RoboDK station: kr30 cnc template 7 axis.rdk

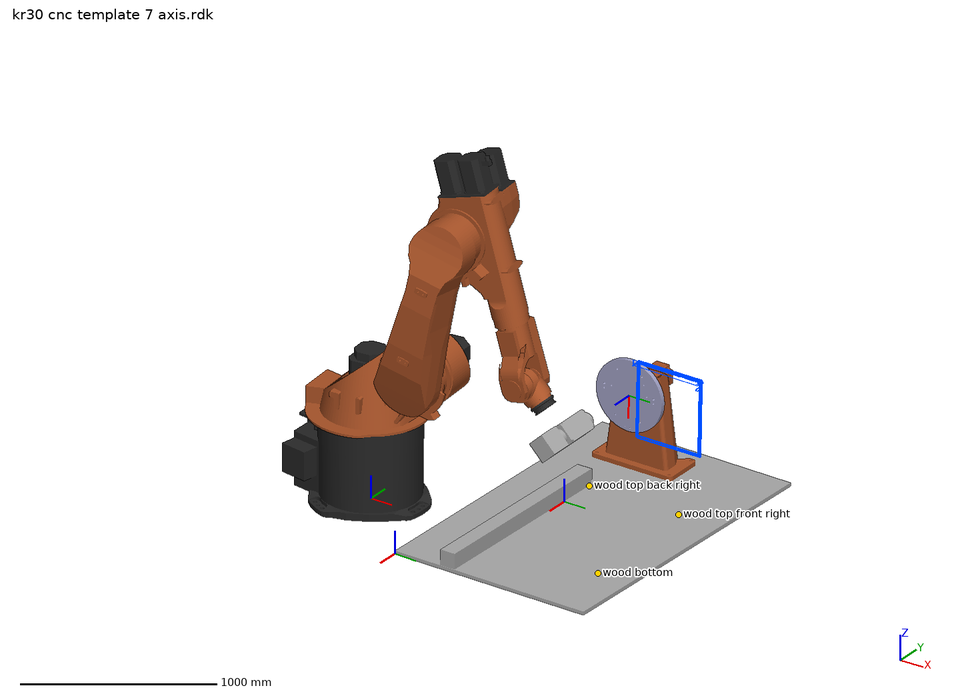
[picture v0: the station drawn from its stored meshes, robots at their saved joint values, targets as dots, program paths as lines]
Station kr30 cnc template 7 axis. Poses are relative to the parent item; angles as X-Y-Z fixed-axis rotations.
  - frame KUKA KR 30 HA Base at (0, 0, 0) mm
    - robot KUKA KR 30 HA: 6 axes, payload 30 kg, reach 2033 mm, repeatability 0.05 mm, weight 665 kg
        modified DH rows (alpha deg, a mm, theta deg, d mm): 0, 0, 0, 815; -90, 350, 0, 0; 0, 850, -90, 0; -90, 145, 0, 820; 90, 0, 0, 0; -90, 0, 180, 170
        joint limits [-185, -135, -120, -350, -119, -350] to [185, 35, 158, 350, 119, 350]; home [0, -90, 90, 0, 0, 0]; saved at [-4.811, -75.793, 150.38, -184.712, 27.792, 91.719]
      - tool rc90 spindle mm, TCP at (267.95, 0.68, 160.99) mm, rotated rx 0 ry 90 rz 0 deg, size 110 x 421.3 x 118 mm, geometry from rc90 spindle mm.stl
    - frame Tabletop at (921.82, -1104.91, 385) mm, rotated rx -0.93 ry -0.21 rz -89.9 deg
      - object tabletop CHECK HEIGHT at (-1839.9, 0, 0) mm, size 1839.9 x 1168.4 x 19 mm, geometry from kr30 tabletop mm.stl
      - object kr30 pipe jig base at (-1220, -610.6, 0) mm, size 1217.6 x 88.9 x 88.9 mm, geometry from kr30 pipe jig base.stl
      - frame Frame 3 at (-930, 400, 45) mm
      - target wood top back right (Cartesian target) at (-1141.49, 406.84, 52.26) mm, rotated rx 18.07 ry 89.88 rz 108.17 deg; joints [-2.086, -55.392, 143.759, 178.106, 87.553, -179.775] of KUKA KR 30 HA
      - target wood bottom (Cartesian target) at (-376.62, 995.52, 35.89) mm, rotated rx 18.07 ry 89.88 rz 108.17 deg; joints [24.587, -27.296, 76.752, 211.623, 53.064, -199.759] of KUKA KR 30 HA
      - target wood top front right (Cartesian target) at (-1142.68, 960.22, 52.55) mm, rotated rx 18.06 ry 89.88 rz 108.16 deg; joints [-1.42, -37.516, 98.016, 178.579, 59.693, -179.129] of KUKA KR 30 HA
  - machining project Machining Settings: C:/Users/Research Office/Desktop/paulina a5.apt | rotZ(0) | rotX(0)*rotY(0) | rotZ(0)
  - frame KUKA KP1 MD250 Base at (1360.87, 339.35, 824.43) mm, rotated rx -93.1 ry 88.62 rz 178.42 deg
    - robot KUKA KP1 MD250: 1 axes, payload 250 kg
        modified DH rows (alpha deg, a mm, theta deg, d mm): 0, 0, 0, 0
        joint limits [-180] to [180]; home [0]; saved at [179]
  - program Machining (2349 instructions, listed below)
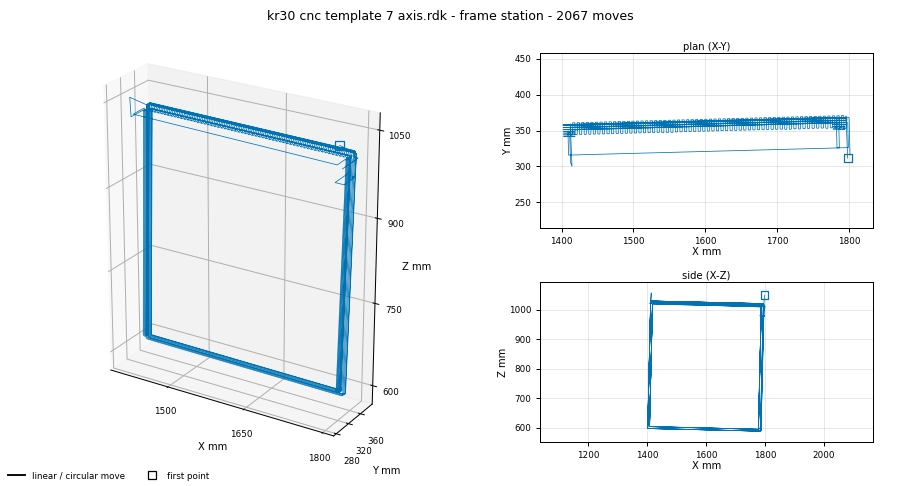
[picture p0: tool path of kr30 cnc template 7 axis.rdk in frame station, 2067 of 2067 moves have a stored position in this frame; points joined in program order, loops and branches not executed]

--- program Machining (robot KUKA KR 30 HA) ---
  Smooth(10)
  Print: /'1001'
  Print: /''
  Print: /'diagonal cut'
  Set speed (100.0 mm/s)
  Set Ref.: KUKA KP1 MD250 Base
  Set Tool: rc90 spindle mm
  Show rc90 spindle mm
  MoveJ 1 to (-235.36, 431, 39.15) mm, rotated rx 174.64 ry -29.65 rz 10.73 deg; joints [4.697, -25.984, 119.452, -143.243, 76.126, 76.923, 151.362]
  MoveL 2 to (-235.36, 431, 39.15) mm, rotated rx 174.64 ry -29.65 rz 10.73 deg; joints [4.697, -25.984, 119.452, -143.243, 76.126, 76.923, 151.362]
  MoveL 3 to (-235.36, 431, 39.15) mm, rotated rx 174.64 ry -29.65 rz 10.73 deg; joints [4.697, -25.984, 119.452, -143.243, 76.126, 76.923, 151.362]
  Set speed (100.0 mm/s)
  MoveL 4 to (-206.65, 431, -10.41) mm, rotated rx 176.37 ry -29.88 rz 7.26 deg; joints [2.395, -27.489, 120.205, -145.105, 75.237, 77.791, 154.384]
  Set speed (38.1 mm/s)
  MoveL 5 to (-201.55, 431, -19.21) mm, rotated rx 176.68 ry -29.92 rz 6.62 deg; joints [1.985, -27.751, 120.32, -145.443, 75.061, 77.953, 154.937]
  MoveL 6 to (-200.68, 431, -19.44) mm, rotated rx 176.74 ry -29.92 rz 6.52 deg; joints [1.975, -27.795, 120.334, -145.44, 75.025, 77.98, 155.032]
  Set speed (76.2 mm/s)
  MoveL 7 to (-202.44, 431, -12.48) mm, rotated rx 176.63 ry -29.91 rz 6.74 deg; joints [2.302, -27.702, 120.276, -145.137, 75.068, 77.922, 154.841]
  MoveL 8 to (-201.13, 431, -12.23) mm, rotated rx 176.71 ry -29.92 rz 6.57 deg; joints [2.315, -27.767, 120.293, -145.106, 75.011, 77.962, 154.983]
  MoveL 9 to (-196.56, 431, -16.91) mm, rotated rx 177 ry -29.95 rz 5.99 deg; joints [2.098, -27.998, 120.38, -145.259, 74.837, 78.109, 155.484]
  Set speed (38.1 mm/s)
  MoveL 10 to (-196.33, 431, -16.04) mm, rotated rx 177.01 ry -29.95 rz 5.97 deg; joints [2.14, -28.009, 120.379, -145.215, 74.823, 78.115, 155.51]
  Set speed (100.0 mm/s)
  MoveL 11 to (-203.65, 431, -3.41) mm, rotated rx 176.55 ry -29.9 rz 6.89 deg; joints [2.729, -27.635, 120.211, -144.726, 75.075, 77.876, 154.709]
  MoveL 12 to (-199.05, 427.82, -0.75) mm, rotated rx 176.75 ry -29.92 rz 6.5 deg; joints [2.857, -28.037, 120.362, -144.533, 74.826, 77.893, 155.049]
  Set speed (38.1 mm/s)
  MoveL 13 to (-197.47, 427.82, -3.47) mm, rotated rx 176.85 ry -29.93 rz 6.3 deg; joints [2.73, -28.118, 120.4, -144.638, 74.772, 77.946, 155.223]
  MoveL 14 to (-197.39, 427.82, -3.84) mm, rotated rx 176.85 ry -29.93 rz 6.29 deg; joints [2.713, -28.123, 120.403, -144.654, 74.77, 77.949, 155.232]
  Set speed (76.2 mm/s)
  MoveL 15 to (-197.71, 427.82, -8.22) mm, rotated rx 176.83 ry -29.93 rz 6.33 deg; joints [2.506, -28.11, 120.422, -144.867, 74.805, 77.944, 155.197]
  MoveL 16 to (-199.91, 427.82, -8.42) mm, rotated rx 176.69 ry -29.92 rz 6.61 deg; joints [2.494, -28, 120.393, -144.91, 74.901, 77.876, 154.954]
  MoveL 17 to (-206.05, 427.82, -11.57) mm, rotated rx 176.31 ry -29.88 rz 7.38 deg; joints [2.339, -27.694, 120.323, -145.155, 75.18, 77.69, 154.283]
  MoveL 18 to (-201.08, 427.82, -20.25) mm, rotated rx 176.62 ry -29.91 rz 6.75 deg; joints [1.934, -27.95, 120.434, -145.489, 75.005, 77.848, 154.826]
  MoveL 19 to (-201.08, 424.65, -20.25) mm, rotated rx 176.53 ry -29.9 rz 6.94 deg; joints [1.933, -28.124, 120.536, -145.493, 74.966, 77.727, 154.662]
  MoveL 20 to (-206.05, 424.65, -11.57) mm, rotated rx 176.21 ry -29.87 rz 7.57 deg; joints [2.337, -27.867, 120.426, -145.161, 75.142, 77.569, 154.116]
  MoveL 21 to (-200.05, 424.65, -8.41) mm, rotated rx 176.59 ry -29.91 rz 6.81 deg; joints [2.493, -28.167, 120.493, -144.915, 74.868, 77.75, 154.775]
  MoveL 22 to (-197.85, 424.65, -8.4) mm, rotated rx 176.73 ry -29.92 rz 6.53 deg; joints [2.496, -28.278, 120.523, -144.88, 74.772, 77.818, 155.019]
  MoveL 23 to (-197.85, 424.65, -4.14) mm, rotated rx 176.73 ry -29.92 rz 6.53 deg; joints [2.697, -28.275, 120.5, -144.678, 74.752, 77.813, 155.019]
  Set speed (38.1 mm/s)
  MoveL 24 to (-197.89, 424.65, -3.98) mm, rotated rx 176.73 ry -29.92 rz 6.54 deg; joints [2.704, -28.273, 120.498, -144.671, 74.753, 77.812, 155.014]
  MoveL 25 to (-198.05, 424.33, -3.7) mm, rotated rx 176.71 ry -29.92 rz 6.58 deg; joints [2.717, -28.282, 120.505, -144.661, 74.754, 77.794, 154.98]
  Set speed (76.2 mm/s)
  MoveL 26 to (-198.05, 421.79, -3.7) mm, rotated rx 176.63 ry -29.91 rz 6.73 deg; joints [2.716, -28.421, 120.586, -144.664, 74.722, 77.696, 154.848]
  Set speed (38.1 mm/s)
  MoveL 27 to (-197.89, 421.47, -3.98) mm, rotated rx 176.63 ry -29.91 rz 6.73 deg; joints [2.703, -28.447, 120.599, -144.674, 74.713, 77.689, 154.849]
  MoveL 28 to (-197.85, 421.47, -4.14) mm, rotated rx 176.64 ry -29.91 rz 6.72 deg; joints [2.695, -28.449, 120.601, -144.681, 74.712, 77.69, 154.854]
  Set speed (76.2 mm/s)
  MoveL 29 to (-197.85, 421.47, -8.28) mm, rotated rx 176.64 ry -29.91 rz 6.72 deg; joints [2.5, -28.452, 120.623, -144.878, 74.732, 77.696, 154.854]
  MoveL 30 to (-200, 421.47, -8.41) mm, rotated rx 176.5 ry -29.9 rz 7 deg; joints [2.492, -28.344, 120.595, -144.919, 74.826, 77.629, 154.614]
  MoveL 31 to (-206.05, 421.47, -11.57) mm, rotated rx 176.12 ry -29.85 rz 7.76 deg; joints [2.335, -28.039, 120.528, -145.168, 75.105, 77.447, 153.947]
  MoveL 32 to (-201.08, 421.47, -20.25) mm, rotated rx 176.43 ry -29.89 rz 7.13 deg; joints [1.931, -28.298, 120.638, -145.498, 74.927, 77.606, 154.495]
  MoveL 33 to (-201.08, 418.3, -20.25) mm, rotated rx 176.33 ry -29.88 rz 7.33 deg; joints [1.929, -28.471, 120.739, -145.503, 74.888, 77.483, 154.326]
  MoveL 34 to (-206.05, 418.3, -11.57) mm, rotated rx 176.02 ry -29.84 rz 7.96 deg; joints [2.333, -28.211, 120.63, -145.175, 75.068, 77.325, 153.776]
  MoveL 35 to (-199.95, 418.3, -8.41) mm, rotated rx 176.41 ry -29.89 rz 7.18 deg; joints [2.49, -28.52, 120.696, -144.922, 74.785, 77.507, 154.452]
  MoveL 36 to (-197.85, 418.3, -8.16) mm, rotated rx 176.54 ry -29.9 rz 6.91 deg; joints [2.504, -28.626, 120.723, -144.876, 74.691, 77.572, 154.687]
  MoveL 37 to (-197.85, 418.3, -4.14) mm, rotated rx 176.54 ry -29.9 rz 6.91 deg; joints [2.694, -28.623, 120.702, -144.685, 74.672, 77.567, 154.687]
  Set speed (38.1 mm/s)
  MoveL 38 to (-197.89, 418.3, -3.98) mm, rotated rx 176.54 ry -29.9 rz 6.92 deg; joints [2.701, -28.621, 120.7, -144.678, 74.673, 77.565, 154.682]
  MoveL 39 to (-198.05, 417.98, -3.7) mm, rotated rx 176.52 ry -29.9 rz 6.96 deg; joints [2.714, -28.63, 120.706, -144.668, 74.675, 77.548, 154.647]
  Set speed (76.2 mm/s)
  MoveL 40 to (-198.05, 415.44, -3.7) mm, rotated rx 176.44 ry -29.89 rz 7.11 deg; joints [2.712, -28.768, 120.787, -144.672, 74.644, 77.448, 154.512]
  Set speed (38.1 mm/s)
  MoveL 41 to (-197.89, 415.12, -3.98) mm, rotated rx 176.44 ry -29.89 rz 7.11 deg; joints [2.699, -28.794, 120.8, -144.683, 74.634, 77.441, 154.513]
  MoveL 42 to (-197.85, 415.12, -4.14) mm, rotated rx 176.44 ry -29.89 rz 7.11 deg; joints [2.692, -28.796, 120.802, -144.689, 74.633, 77.443, 154.518]
  Set speed (76.2 mm/s)
  MoveL 43 to (-197.85, 415.12, -8.4) mm, rotated rx 176.44 ry -29.89 rz 7.11 deg; joints [2.491, -28.8, 120.825, -144.892, 74.653, 77.448, 154.518]
  MoveL 44 to (-199.9, 415.12, -8.41) mm, rotated rx 176.31 ry -29.88 rz 7.37 deg; joints [2.488, -28.695, 120.798, -144.927, 74.744, 77.385, 154.288]
  MoveL 45 to (-206.05, 415.12, -11.57) mm, rotated rx 175.92 ry -29.83 rz 8.16 deg; joints [2.331, -28.382, 120.732, -145.182, 75.031, 77.201, 153.602]
  MoveL 46 to (-201.08, 415.12, -20.25) mm, rotated rx 176.24 ry -29.87 rz 7.53 deg; joints [1.927, -28.643, 120.84, -145.509, 74.849, 77.36, 154.155]
  MoveL 47 to (-201.08, 411.95, -20.25) mm, rotated rx 176.14 ry -29.86 rz 7.72 deg; joints [1.925, -28.816, 120.94, -145.515, 74.81, 77.235, 153.982]
  MoveL 48 to (-206.05, 411.95, -11.57) mm, rotated rx 175.82 ry -29.82 rz 8.36 deg; joints [2.329, -28.553, 120.833, -145.19, 74.995, 77.077, 153.427]
  MoveL 49 to (-199.84, 411.95, -8.41) mm, rotated rx 176.22 ry -29.87 rz 7.56 deg; joints [2.486, -28.87, 120.899, -144.931, 74.703, 77.262, 154.121]
  MoveL 50 to (-197.85, 411.95, -8.4) mm, rotated rx 176.35 ry -29.88 rz 7.31 deg; joints [2.489, -28.973, 120.925, -144.897, 74.614, 77.323, 154.346]
  MoveL 51 to (-197.85, 411.95, -4.14) mm, rotated rx 176.35 ry -29.88 rz 7.31 deg; joints [2.69, -28.969, 120.902, -144.694, 74.594, 77.317, 154.346]
  Set speed (38.1 mm/s)
  MoveL 52 to (-197.89, 411.95, -3.98) mm, rotated rx 176.34 ry -29.88 rz 7.31 deg; joints [2.698, -28.967, 120.9, -144.687, 74.595, 77.316, 154.342]
  MoveL 53 to (-198.05, 411.63, -3.7) mm, rotated rx 176.32 ry -29.88 rz 7.35 deg; joints [2.71, -28.976, 120.907, -144.678, 74.597, 77.298, 154.306]
  Set speed (76.2 mm/s)
  MoveL 54 to (-198.05, 409.09, -3.7) mm, rotated rx 176.24 ry -29.87 rz 7.51 deg; joints [2.709, -29.114, 120.986, -144.682, 74.566, 77.197, 154.168]
  Set speed (38.1 mm/s)
  MoveL 55 to (-197.89, 408.77, -3.98) mm, rotated rx 176.24 ry -29.87 rz 7.51 deg; joints [2.696, -29.139, 121, -144.693, 74.557, 77.19, 154.168]
  MoveL 56 to (-197.85, 408.77, -4.14) mm, rotated rx 176.25 ry -29.87 rz 7.5 deg; joints [2.688, -29.141, 121.001, -144.7, 74.555, 77.191, 154.173]
  Set speed (76.2 mm/s)
  MoveL 57 to (-197.85, 408.77, -8.4) mm, rotated rx 176.25 ry -29.87 rz 7.5 deg; joints [2.487, -29.145, 121.024, -144.903, 74.575, 77.197, 154.173]
  MoveL 58 to (-200.19, 408.77, -8.41) mm, rotated rx 176.09 ry -29.85 rz 7.81 deg; joints [2.484, -29.024, 120.994, -144.944, 74.681, 77.125, 153.907]
  MoveL 59 to (-206.05, 408.77, -11.57) mm, rotated rx 175.72 ry -29.8 rz 8.57 deg; joints [2.326, -28.724, 120.934, -145.199, 74.958, 76.952, 153.249]
  MoveL 60 to (-201.08, 408.77, -20.25) mm, rotated rx 176.04 ry -29.84 rz 7.93 deg; joints [1.923, -28.987, 121.041, -145.522, 74.772, 77.11, 153.807]
  MoveL 61 to (-201.08, 405.6, -20.25) mm, rotated rx 175.94 ry -29.83 rz 8.13 deg; joints [1.92, -29.159, 121.14, -145.53, 74.734, 76.984, 153.63]
  MoveL 62 to (-206.05, 405.6, -11.57) mm, rotated rx 175.61 ry -29.79 rz 8.77 deg; joints [2.324, -28.894, 121.035, -145.208, 74.922, 76.826, 153.069]
  MoveL 63 to (-200.12, 405.6, -8.41) mm, rotated rx 176 ry -29.84 rz 8 deg; joints [2.482, -29.199, 121.095, -144.95, 74.64, 77.001, 153.738]
  MoveL 64 to (-197.85, 405.6, -8.4) mm, rotated rx 176.15 ry -29.86 rz 7.71 deg; joints [2.485, -29.317, 121.124, -144.909, 74.536, 77.071, 153.997]
  MoveL 65 to (-197.85, 405.6, -4.14) mm, rotated rx 176.15 ry -29.86 rz 7.71 deg; joints [2.686, -29.313, 121.101, -144.706, 74.517, 77.065, 153.997]
  MoveL 66 to (-197.85, 405.47, -3.66) mm, rotated rx 176.14 ry -29.86 rz 7.71 deg; joints [2.709, -29.32, 121.102, -144.683, 74.513, 77.059, 153.99]
  MoveL 67 to (-197.85, 405.12, -3.31) mm, rotated rx 176.13 ry -29.86 rz 7.74 deg; joints [2.725, -29.338, 121.111, -144.667, 74.507, 77.044, 153.971]
  MoveL 68 to (-197.85, 404.64, -3.19) mm, rotated rx 176.12 ry -29.85 rz 7.77 deg; joints [2.731, -29.364, 121.125, -144.662, 74.501, 77.025, 153.944]
  MoveL 69 to (-197.85, 403.38, -3.19) mm, rotated rx 176.07 ry -29.85 rz 7.85 deg; joints [2.73, -29.433, 121.165, -144.665, 74.486, 76.974, 153.873]
  MoveL 70 to (-197.85, 402.9, -3.31) mm, rotated rx 176.06 ry -29.85 rz 7.88 deg; joints [2.723, -29.458, 121.18, -144.672, 74.481, 76.955, 153.846]
  MoveL 71 to (-197.85, 402.55, -3.66) mm, rotated rx 176.05 ry -29.85 rz 7.9 deg; joints [2.707, -29.477, 121.193, -144.689, 74.478, 76.941, 153.827]
  MoveL 72 to (-197.85, 402.42, -4.14) mm, rotated rx 176.04 ry -29.85 rz 7.91 deg; joints [2.684, -29.485, 121.199, -144.712, 74.479, 76.937, 153.82]
  MoveL 73 to (-197.85, 402.42, -8.4) mm, rotated rx 176.04 ry -29.85 rz 7.91 deg; joints [2.483, -29.488, 121.222, -144.915, 74.498, 76.943, 153.82]
  MoveL 74 to (-200.05, 402.42, -8.41) mm, rotated rx 175.9 ry -29.83 rz 8.2 deg; joints [2.48, -29.374, 121.195, -144.956, 74.599, 76.876, 153.567]
  MoveL 75 to (-206.05, 402.42, -11.57) mm, rotated rx 175.51 ry -29.78 rz 8.98 deg; joints [2.321, -29.063, 121.135, -145.218, 74.887, 76.699, 152.887]
  MoveL 76 to (-201.08, 402.42, -20.25) mm, rotated rx 175.83 ry -29.82 rz 8.34 deg; joints [1.918, -29.329, 121.24, -145.538, 74.697, 76.858, 153.45]
  MoveL 77 to (-201.08, 399.25, -20.25) mm, rotated rx 175.73 ry -29.81 rz 8.55 deg; joints [1.916, -29.499, 121.339, -145.547, 74.659, 76.73, 153.268]
  MoveL 78 to (-206.05, 399.25, -11.57) mm, rotated rx 175.41 ry -29.76 rz 9.2 deg; joints [2.319, -29.232, 121.235, -145.229, 74.852, 76.572, 152.702]
  MoveL 79 to (-199.98, 399.25, -8.41) mm, rotated rx 175.8 ry -29.82 rz 8.4 deg; joints [2.477, -29.548, 121.295, -144.963, 74.559, 76.75, 153.394]
  MoveL 80 to (-197.85, 399.25, -8.4) mm, rotated rx 175.94 ry -29.83 rz 8.12 deg; joints [2.481, -29.659, 121.321, -144.923, 74.46, 76.815, 153.64]
  MoveL 81 to (-197.85, 399.25, -4.14) mm, rotated rx 175.94 ry -29.83 rz 8.12 deg; joints [2.682, -29.656, 121.298, -144.72, 74.441, 76.808, 153.64]
  Set speed (38.1 mm/s)
  MoveL 82 to (-197.89, 399.25, -3.98) mm, rotated rx 175.94 ry -29.83 rz 8.12 deg; joints [2.69, -29.653, 121.297, -144.713, 74.442, 76.807, 153.635]
  MoveL 83 to (-198.05, 398.93, -3.7) mm, rotated rx 175.92 ry -29.83 rz 8.17 deg; joints [2.702, -29.662, 121.303, -144.704, 74.444, 76.789, 153.598]
  Set speed (76.2 mm/s)
  MoveL 84 to (-198.05, 396.39, -3.7) mm, rotated rx 175.83 ry -29.82 rz 8.33 deg; joints [2.7, -29.798, 121.382, -144.71, 74.415, 76.685, 153.452]
  Set speed (38.1 mm/s)
  MoveL 85 to (-197.89, 396.07, -3.98) mm, rotated rx 175.83 ry -29.82 rz 8.33 deg; joints [2.687, -29.823, 121.395, -144.721, 74.405, 76.677, 153.452]
  MoveL 86 to (-197.85, 396.07, -4.14) mm, rotated rx 175.84 ry -29.82 rz 8.33 deg; joints [2.68, -29.826, 121.396, -144.728, 74.403, 76.679, 153.457]
  Set speed (76.2 mm/s)
  MoveL 87 to (-197.85, 396.07, -8.4) mm, rotated rx 175.84 ry -29.82 rz 8.33 deg; joints [2.479, -29.829, 121.419, -144.931, 74.422, 76.686, 153.457]
  MoveL 88 to (-199.91, 396.07, -8.41) mm, rotated rx 175.7 ry -29.8 rz 8.6 deg; joints [2.475, -29.721, 121.394, -144.971, 74.518, 76.623, 153.218]
  MoveL 89 to (-206.05, 396.07, -11.57) mm, rotated rx 175.3 ry -29.75 rz 9.41 deg; joints [2.316, -29.4, 121.335, -145.241, 74.817, 76.443, 152.515]
  MoveL 90 to (-201.08, 396.07, -20.25) mm, rotated rx 175.62 ry -29.79 rz 8.76 deg; joints [1.913, -29.669, 121.438, -145.557, 74.622, 76.602, 153.084]
  MoveL 91 to (-201.08, 392.9, -20.25) mm, rotated rx 175.52 ry -29.78 rz 8.97 deg; joints [1.91, -29.838, 121.536, -145.567, 74.586, 76.473, 152.898]
  MoveL 92 to (-206.05, 392.9, -11.57) mm, rotated rx 175.19 ry -29.73 rz 9.63 deg; joints [2.313, -29.568, 121.434, -145.253, 74.782, 76.314, 152.326]
  MoveL 93 to (-199.84, 392.9, -8.41) mm, rotated rx 175.6 ry -29.79 rz 8.81 deg; joints [2.473, -29.894, 121.493, -144.979, 74.479, 76.495, 153.04]
  MoveL 94 to (-197.85, 392.9, -8.38) mm, rotated rx 175.73 ry -29.81 rz 8.54 deg; joints [2.477, -29.999, 121.517, -144.938, 74.385, 76.556, 153.272]
  MoveL 95 to (-197.85, 392.9, -4.14) mm, rotated rx 175.73 ry -29.81 rz 8.54 deg; joints [2.677, -29.996, 121.494, -144.736, 74.366, 76.549, 153.272]
  Set speed (38.1 mm/s)
  MoveL 96 to (-197.89, 392.9, -3.98) mm, rotated rx 175.73 ry -29.81 rz 8.55 deg; joints [2.685, -29.993, 121.493, -144.729, 74.368, 76.547, 153.267]
  MoveL 97 to (-198.05, 392.58, -3.7) mm, rotated rx 175.71 ry -29.8 rz 8.59 deg; joints [2.697, -30.002, 121.499, -144.72, 74.37, 76.529, 153.23]
  Set speed (76.2 mm/s)
  MoveL 98 to (-198.05, 390.04, -3.7) mm, rotated rx 175.62 ry -29.79 rz 8.76 deg; joints [2.695, -30.137, 121.577, -144.728, 74.341, 76.424, 153.08]
  Set speed (38.1 mm/s)
  MoveL 99 to (-197.89, 389.72, -3.98) mm, rotated rx 175.62 ry -29.79 rz 8.76 deg; joints [2.682, -30.162, 121.59, -144.739, 74.331, 76.416, 153.08]
  MoveL 100 to (-197.85, 389.72, -4.14) mm, rotated rx 175.62 ry -29.79 rz 8.76 deg; joints [2.675, -30.165, 121.592, -144.746, 74.329, 76.418, 153.085]
  Set speed (76.2 mm/s)
  MoveL 101 to (-197.85, 389.72, -8.26) mm, rotated rx 175.62 ry -29.79 rz 8.76 deg; joints [2.48, -30.168, 121.614, -144.942, 74.348, 76.425, 153.085]
  MoveL 102 to (-199.77, 389.72, -8.41) mm, rotated rx 175.5 ry -29.77 rz 9.01 deg; joints [2.47, -30.066, 121.592, -144.988, 74.439, 76.366, 152.86]
  MoveL 103 to (-206.05, 389.72, -11.57) mm, rotated rx 175.08 ry -29.71 rz 9.85 deg; joints [2.31, -29.736, 121.533, -145.266, 74.748, 76.184, 152.134]
  MoveL 104 to (-201.08, 389.72, -20.25) mm, rotated rx 175.41 ry -29.76 rz 9.19 deg; joints [1.908, -30.007, 121.634, -145.578, 74.549, 76.343, 152.709]
  MoveL 105 to (-201.08, 386.55, -20.25) mm, rotated rx 175.3 ry -29.75 rz 9.41 deg; joints [1.905, -30.175, 121.732, -145.59, 74.513, 76.212, 152.517]
  MoveL 106 to (-206.05, 386.55, -11.57) mm, rotated rx 174.97 ry -29.7 rz 10.07 deg; joints [2.307, -29.902, 121.632, -145.279, 74.714, 76.053, 151.94]
  MoveL 107 to (-199.7, 386.55, -8.41) mm, rotated rx 175.39 ry -29.76 rz 9.22 deg; joints [2.467, -30.238, 121.69, -144.997, 74.4, 76.237, 152.678]
  MoveL 108 to (-197.85, 386.55, -8.41) mm, rotated rx 175.52 ry -29.78 rz 8.97 deg; joints [2.471, -30.337, 121.712, -144.959, 74.312, 76.293, 152.896]
  MoveL 109 to (-197.85, 386.55, -4.14) mm, rotated rx 175.52 ry -29.78 rz 8.97 deg; joints [2.672, -30.334, 121.689, -144.756, 74.293, 76.286, 152.896]
  Set speed (38.1 mm/s)
  MoveL 110 to (-197.89, 386.55, -3.98) mm, rotated rx 175.51 ry -29.78 rz 8.98 deg; joints [2.68, -30.331, 121.688, -144.749, 74.294, 76.284, 152.89]
  MoveL 111 to (-198.05, 386.23, -3.7) mm, rotated rx 175.49 ry -29.77 rz 9.02 deg; joints [2.692, -30.339, 121.694, -144.74, 74.297, 76.266, 152.853]
  Set speed (76.2 mm/s)
  MoveL 112 to (-198.05, 383.69, -3.7) mm, rotated rx 175.4 ry -29.76 rz 9.2 deg; joints [2.69, -30.474, 121.772, -144.749, 74.268, 76.16, 152.699]
  Set speed (38.1 mm/s)
  MoveL 113 to (-197.89, 383.37, -3.98) mm, rotated rx 175.4 ry -29.76 rz 9.2 deg; joints [2.677, -30.499, 121.785, -144.76, 74.258, 76.152, 152.698]
  MoveL 114 to (-197.85, 383.37, -4.14) mm, rotated rx 175.41 ry -29.76 rz 9.19 deg; joints [2.67, -30.502, 121.786, -144.767, 74.257, 76.153, 152.703]
  Set speed (76.2 mm/s)
  MoveL 115 to (-197.85, 383.37, -8.4) mm, rotated rx 175.41 ry -29.76 rz 9.19 deg; joints [2.468, -30.505, 121.809, -144.97, 74.275, 76.161, 152.703]
  MoveL 116 to (-199.66, 383.37, -8.41) mm, rotated rx 175.28 ry -29.74 rz 9.44 deg; joints [2.465, -30.409, 121.788, -145.008, 74.362, 76.106, 152.49]
  MoveL 117 to (-206.05, 383.37, -11.57) mm, rotated rx 174.86 ry -29.68 rz 10.3 deg; joints [2.304, -30.068, 121.731, -145.294, 74.68, 75.922, 151.744]
  MoveL 118 to (-201.08, 383.37, -20.25) mm, rotated rx 175.19 ry -29.73 rz 9.63 deg; joints [1.902, -30.342, 121.83, -145.603, 74.478, 76.08, 152.323]
  MoveL 119 to (-201.08, 380.2, -20.25) mm, rotated rx 175.08 ry -29.71 rz 9.86 deg; joints [1.898, -30.509, 121.927, -145.616, 74.443, 75.947, 152.127]
  MoveL 120 to (-206.05, 380.2, -11.57) mm, rotated rx 174.75 ry -29.66 rz 10.52 deg; joints [2.3, -30.234, 121.829, -145.309, 74.647, 75.789, 151.545]
  MoveL 121 to (-200.12, 380.2, -8.41) mm, rotated rx 175.14 ry -29.72 rz 9.73 deg; joints [2.461, -30.551, 121.88, -145.03, 74.349, 75.959, 152.24]
  MoveL 122 to (-197.85, 380.2, -8.4) mm, rotated rx 175.3 ry -29.75 rz 9.42 deg; joints [2.465, -30.673, 121.906, -144.982, 74.239, 76.027, 152.509]
  MoveL 123 to (-197.85, 380.2, -4.14) mm, rotated rx 175.3 ry -29.75 rz 9.42 deg; joints [2.667, -30.669, 121.883, -144.778, 74.221, 76.02, 152.509]
  Set speed (38.1 mm/s)
  MoveL 124 to (-197.89, 380.2, -3.98) mm, rotated rx 175.29 ry -29.75 rz 9.42 deg; joints [2.674, -30.667, 121.881, -144.771, 74.223, 76.018, 152.504]
  MoveL 125 to (-198.05, 379.88, -3.7) mm, rotated rx 175.27 ry -29.74 rz 9.47 deg; joints [2.687, -30.675, 121.888, -144.763, 74.226, 75.999, 152.465]
  Set speed (76.2 mm/s)
  MoveL 126 to (-198.05, 377.34, -3.7) mm, rotated rx 175.18 ry -29.73 rz 9.65 deg; joints [2.684, -30.808, 121.965, -144.773, 74.197, 75.892, 152.307]
  Set speed (38.1 mm/s)
  MoveL 127 to (-197.89, 377.02, -3.98) mm, rotated rx 175.18 ry -29.73 rz 9.65 deg; joints [2.671, -30.834, 121.978, -144.784, 74.187, 75.884, 152.306]
  MoveL 128 to (-197.85, 377.02, -4.14) mm, rotated rx 175.18 ry -29.73 rz 9.64 deg; joints [2.664, -30.836, 121.979, -144.791, 74.186, 75.885, 152.312]
  Set speed (76.2 mm/s)
  MoveL 129 to (-197.85, 377.02, -8.4) mm, rotated rx 175.18 ry -29.73 rz 9.64 deg; joints [2.462, -30.84, 122.002, -144.994, 74.204, 75.893, 152.312]
  MoveL 130 to (-200.07, 377.02, -8.41) mm, rotated rx 175.03 ry -29.71 rz 9.95 deg; joints [2.458, -30.72, 121.978, -145.043, 74.312, 75.827, 152.048]
  MoveL 131 to (-206.05, 377.02, -11.57) mm, rotated rx 174.63 ry -29.64 rz 10.75 deg; joints [2.297, -30.399, 121.927, -145.326, 74.615, 75.656, 151.343]
  MoveL 132 to (-201.08, 377.02, -20.25) mm, rotated rx 174.96 ry -29.7 rz 10.08 deg; joints [1.895, -30.675, 122.024, -145.63, 74.408, 75.814, 151.928]
  MoveL 133 to (-201.08, 373.85, -20.25) mm, rotated rx 174.85 ry -29.68 rz 10.32 deg; joints [1.892, -30.841, 122.121, -145.646, 74.374, 75.68, 151.726]
  MoveL 134 to (-206.05, 373.85, -11.57) mm, rotated rx 174.52 ry -29.62 rz 10.99 deg; joints [2.293, -30.564, 122.025, -145.343, 74.582, 75.522, 151.138]
  MoveL 135 to (-200.58, 373.85, -8.41) mm, rotated rx 174.88 ry -29.68 rz 10.25 deg; joints [2.454, -30.858, 122.069, -145.069, 74.303, 75.677, 151.785]
  MoveL 136 to (-197.85, 373.85, -8.4) mm, rotated rx 175.07 ry -29.71 rz 9.87 deg; joints [2.459, -31.006, 122.098, -145.008, 74.169, 75.758, 152.112]
  MoveL 137 to (-197.85, 373.85, -4.14) mm, rotated rx 175.07 ry -29.71 rz 9.87 deg; joints [2.661, -31.003, 122.076, -144.804, 74.151, 75.75, 152.112]
  Set speed (38.1 mm/s)
  MoveL 138 to (-197.89, 373.85, -3.98) mm, rotated rx 175.07 ry -29.71 rz 9.88 deg; joints [2.668, -31, 122.074, -144.797, 74.153, 75.748, 152.107]
  MoveL 139 to (-198.05, 373.53, -3.7) mm, rotated rx 175.04 ry -29.71 rz 9.92 deg; joints [2.681, -31.008, 122.081, -144.789, 74.156, 75.729, 152.067]
  Set speed (76.2 mm/s)
  MoveL 140 to (-198.05, 370.99, -3.7) mm, rotated rx 174.95 ry -29.7 rz 10.11 deg; joints [2.678, -31.141, 122.157, -144.8, 74.128, 75.621, 151.905]
  Set speed (38.1 mm/s)
  MoveL 141 to (-197.89, 370.67, -3.98) mm, rotated rx 174.95 ry -29.69 rz 10.11 deg; joints [2.665, -31.166, 122.17, -144.811, 74.118, 75.612, 151.904]
  MoveL 142 to (-197.85, 370.68, -4.14) mm, rotated rx 174.95 ry -29.7 rz 10.11 deg; joints [2.658, -31.168, 122.172, -144.818, 74.117, 75.614, 151.909]
  Set speed (76.2 mm/s)
  MoveL 143 to (-197.85, 370.68, -8.4) mm, rotated rx 174.95 ry -29.7 rz 10.11 deg; joints [2.456, -31.172, 122.194, -145.022, 74.135, 75.622, 151.909]
  MoveL 144 to (-200.55, 370.67, -8.41) mm, rotated rx 174.77 ry -29.67 rz 10.48 deg; joints [2.45, -31.025, 122.166, -145.083, 74.268, 75.542, 151.585]
  MoveL 145 to (-206.05, 370.68, -11.57) mm, rotated rx 174.4 ry -29.6 rz 11.23 deg; joints [2.289, -30.727, 122.123, -145.361, 74.551, 75.387, 150.931]
  MoveL 146 to (-201.08, 370.68, -20.25) mm, rotated rx 174.73 ry -29.66 rz 10.55 deg; joints [1.888, -31.006, 122.218, -145.662, 74.34, 75.545, 151.522]
  MoveL 147 to (-201.08, 367.5, -20.25) mm, rotated rx 174.62 ry -29.64 rz 10.79 deg; joints [1.884, -31.171, 122.314, -145.679, 74.306, 75.409, 151.315]
  MoveL 148 to (-206.05, 367.5, -11.57) mm, rotated rx 174.28 ry -29.58 rz 11.47 deg; joints [2.285, -30.891, 122.22, -145.38, 74.519, 75.252, 150.722]
  MoveL 149 to (-200.51, 367.5, -8.41) mm, rotated rx 174.66 ry -29.65 rz 10.71 deg; joints [2.447, -31.192, 122.263, -145.099, 74.233, 75.407, 151.383]
  MoveL 150 to (-197.85, 367.5, -8.4) mm, rotated rx 174.84 ry -29.68 rz 10.34 deg; joints [2.453, -31.338, 122.29, -145.037, 74.1, 75.485, 151.704]
  MoveL 151 to (-197.85, 367.5, -4.14) mm, rotated rx 174.84 ry -29.68 rz 10.34 deg; joints [2.654, -31.334, 122.267, -144.833, 74.083, 75.477, 151.704]
  MoveL 152 to (-197.85, 367.37, -3.66) mm, rotated rx 174.83 ry -29.68 rz 10.35 deg; joints [2.677, -31.34, 122.269, -144.811, 74.08, 75.47, 151.696]
  MoveL 153 to (-197.85, 367.02, -3.31) mm, rotated rx 174.82 ry -29.67 rz 10.38 deg; joints [2.693, -31.358, 122.277, -144.796, 74.074, 75.455, 151.673]
  MoveL 154 to (-197.85, 366.55, -3.19) mm, rotated rx 174.8 ry -29.67 rz 10.41 deg; joints [2.698, -31.382, 122.291, -144.792, 74.069, 75.434, 151.642]
  MoveL 155 to (-197.85, 365.28, -3.19) mm, rotated rx 174.76 ry -29.66 rz 10.51 deg; joints [2.697, -31.448, 122.329, -144.799, 74.056, 75.379, 151.559]
  MoveL 156 to (-197.85, 364.8, -3.31) mm, rotated rx 174.74 ry -29.66 rz 10.54 deg; joints [2.69, -31.473, 122.344, -144.807, 74.051, 75.358, 151.527]
  MoveL 157 to (-197.85, 364.45, -3.66) mm, rotated rx 174.72 ry -29.66 rz 10.57 deg; joints [2.674, -31.491, 122.357, -144.826, 74.049, 75.344, 151.504]
  MoveL 158 to (-197.85, 364.33, -4.14) mm, rotated rx 174.72 ry -29.66 rz 10.58 deg; joints [2.651, -31.498, 122.363, -144.849, 74.05, 75.339, 151.496]
  MoveL 159 to (-197.85, 364.33, -8.4) mm, rotated rx 174.72 ry -29.66 rz 10.58 deg; joints [2.449, -31.502, 122.386, -145.053, 74.067, 75.348, 151.496]
  MoveL 160 to (-200.48, 364.33, -8.41) mm, rotated rx 174.54 ry -29.63 rz 10.94 deg; joints [2.443, -31.358, 122.359, -145.116, 74.198, 75.27, 151.177]
  MoveL 161 to (-206.05, 364.33, -11.57) mm, rotated rx 174.16 ry -29.56 rz 11.71 deg; joints [2.281, -31.053, 122.317, -145.4, 74.489, 75.115, 150.509]
  MoveL 162 to (-201.08, 364.33, -20.25) mm, rotated rx 174.5 ry -29.62 rz 11.03 deg; joints [1.881, -31.334, 122.41, -145.696, 74.274, 75.272, 151.105]
  MoveL 163 to (-201.08, 361.15, -20.25) mm, rotated rx 174.38 ry -29.6 rz 11.27 deg; joints [1.877, -31.498, 122.507, -145.715, 74.241, 75.135, 150.892]
  MoveL 164 to (-206.05, 361.15, -11.57) mm, rotated rx 174.04 ry -29.54 rz 11.96 deg; joints [2.277, -31.215, 122.415, -145.421, 74.458, 74.978, 150.294]
  MoveL 165 to (-200.44, 361.15, -8.41) mm, rotated rx 174.42 ry -29.61 rz 11.18 deg; joints [2.44, -31.523, 122.455, -145.133, 74.165, 75.133, 150.969]
  MoveL 166 to (-197.85, 361.15, -8.4) mm, rotated rx 174.6 ry -29.64 rz 10.82 deg; joints [2.445, -31.666, 122.481, -145.07, 74.034, 75.209, 151.285]
  MoveL 167 to (-197.85, 361.15, -4.14) mm, rotated rx 174.6 ry -29.64 rz 10.82 deg; joints [2.647, -31.662, 122.458, -144.866, 74.017, 75.201, 151.285]
  Set speed (38.1 mm/s)
  MoveL 168 to (-197.89, 361.15, -3.98) mm, rotated rx 174.6 ry -29.64 rz 10.83 deg; joints [2.655, -31.66, 122.457, -144.859, 74.018, 75.199, 151.28]
  MoveL 169 to (-198.05, 360.83, -3.7) mm, rotated rx 174.57 ry -29.63 rz 10.87 deg; joints [2.667, -31.667, 122.464, -144.852, 74.022, 75.18, 151.239]
  Set speed (76.2 mm/s)
  MoveL 170 to (-198.05, 358.29, -3.7) mm, rotated rx 174.48 ry -29.62 rz 11.07 deg; joints [2.664, -31.798, 122.54, -144.866, 73.996, 75.068, 151.068]
  Set speed (38.1 mm/s)
  MoveL 171 to (-197.89, 357.98, -3.98) mm, rotated rx 174.48 ry -29.62 rz 11.07 deg; joints [2.651, -31.823, 122.552, -144.877, 73.986, 75.06, 151.066]
  MoveL 172 to (-197.85, 357.98, -4.14) mm, rotated rx 174.48 ry -29.62 rz 11.07 deg; joints [2.644, -31.826, 122.554, -144.884, 73.984, 75.061, 151.072]
  Set speed (76.2 mm/s)
  MoveL 173 to (-197.85, 357.98, -8.25) mm, rotated rx 174.48 ry -29.62 rz 11.07 deg; joints [2.449, -31.829, 122.576, -145.081, 74.001, 75.07, 151.072]
  MoveL 174 to (-200.41, 357.98, -8.41) mm, rotated rx 174.3 ry -29.59 rz 11.42 deg; joints [2.436, -31.688, 122.552, -145.152, 74.131, 74.995, 150.758]
  MoveL 175 to (-206.05, 357.98, -11.57) mm, rotated rx 173.92 ry -29.52 rz 12.2 deg; joints [2.273, -31.377, 122.512, -145.443, 74.429, 74.84, 150.076]
  MoveL 176 to (-201.08, 357.98, -20.25) mm, rotated rx 174.26 ry -29.58 rz 11.52 deg; joints [1.872, -31.66, 122.602, -145.735, 74.209, 74.996, 150.677]
  MoveL 177 to (-201.08, 354.8, -20.25) mm, rotated rx 174.13 ry -29.56 rz 11.77 deg; joints [1.868, -31.822, 122.698, -145.756, 74.178, 74.857, 150.458]
  MoveL 178 to (-206.05, 354.8, -11.57) mm, rotated rx 173.79 ry -29.49 rz 12.46 deg; joints [2.268, -31.537, 122.608, -145.466, 74.399, 74.701, 149.854]
  MoveL 179 to (-200.37, 354.8, -8.41) mm, rotated rx 174.18 ry -29.57 rz 11.67 deg; joints [2.432, -31.852, 122.647, -145.171, 74.098, 74.857, 150.544]
  MoveL 180 to (-197.85, 354.8, -8.13) mm, rotated rx 174.36 ry -29.6 rz 11.31 deg; joints [2.451, -31.992, 122.67, -145.094, 73.968, 74.93, 150.855]
  MoveL 181 to (-197.85, 354.8, -4.14) mm, rotated rx 174.36 ry -29.6 rz 11.31 deg; joints [2.64, -31.988, 122.649, -144.903, 73.952, 74.921, 150.855]
  MoveL 182 to (-197.85, 354.67, -3.66) mm, rotated rx 174.35 ry -29.6 rz 11.32 deg; joints [2.662, -31.994, 122.65, -144.881, 73.949, 74.914, 150.846]
  MoveL 183 to (-197.85, 354.33, -3.31) mm, rotated rx 174.34 ry -29.59 rz 11.35 deg; joints [2.678, -32.012, 122.658, -144.866, 73.944, 74.898, 150.822]
  MoveL 184 to (-197.85, 353.85, -3.19) mm, rotated rx 174.32 ry -29.59 rz 11.39 deg; joints [2.684, -32.036, 122.672, -144.863, 73.939, 74.876, 150.789]
  MoveL 185 to (-197.85, 352.58, -3.19) mm, rotated rx 174.27 ry -29.58 rz 11.49 deg; joints [2.682, -32.101, 122.71, -144.871, 73.927, 74.82, 150.702]
  MoveL 186 to (-197.85, 352.1, -3.31) mm, rotated rx 174.25 ry -29.58 rz 11.53 deg; joints [2.675, -32.125, 122.725, -144.88, 73.922, 74.799, 150.669]
  MoveL 187 to (-197.85, 351.75, -3.66) mm, rotated rx 174.24 ry -29.58 rz 11.55 deg; joints [2.658, -32.143, 122.737, -144.899, 73.92, 74.784, 150.644]
  MoveL 188 to (-197.85, 351.63, -4.14) mm, rotated rx 174.23 ry -29.58 rz 11.56 deg; joints [2.636, -32.15, 122.744, -144.923, 73.921, 74.78, 150.635]
  MoveL 189 to (-197.85, 351.63, -8.4) mm, rotated rx 174.23 ry -29.58 rz 11.56 deg; joints [2.433, -32.154, 122.767, -145.128, 73.938, 74.789, 150.635]
  MoveL 190 to (-200.34, 351.63, -8.41) mm, rotated rx 174.06 ry -29.54 rz 11.92 deg; joints [2.427, -32.015, 122.743, -145.192, 74.066, 74.717, 150.328]
  MoveL 191 to (-206.05, 351.63, -11.57) mm, rotated rx 173.67 ry -29.47 rz 12.71 deg; joints [2.263, -31.697, 122.705, -145.491, 74.371, 74.561, 149.63]
  MoveL 192 to (-201.08, 351.63, -20.25) mm, rotated rx 174.01 ry -29.53 rz 12.02 deg; joints [1.864, -31.984, 122.794, -145.778, 74.147, 74.717, 150.237]
  MoveL 193 to (-201.08, 348.45, -20.25) mm, rotated rx 173.88 ry -29.51 rz 12.28 deg; joints [1.859, -32.144, 122.889, -145.802, 74.117, 74.576, 150.012]
  MoveL 194 to (-206.05, 348.45, -11.57) mm, rotated rx 173.54 ry -29.44 rz 12.97 deg; joints [2.258, -31.857, 122.802, -145.516, 74.342, 74.421, 149.403]
  MoveL 195 to (-199.95, 348.45, -8.41) mm, rotated rx 173.96 ry -29.53 rz 12.12 deg; joints [2.424, -32.197, 122.842, -145.204, 74.016, 74.587, 150.151]
  MoveL 196 to (-197.85, 348.45, -8.4) mm, rotated rx 174.11 ry -29.55 rz 11.82 deg; joints [2.429, -32.316, 122.861, -145.149, 73.907, 74.647, 150.413]
  MoveL 197 to (-197.85, 348.45, -4.14) mm, rotated rx 174.11 ry -29.55 rz 11.82 deg; joints [2.631, -32.312, 122.838, -144.944, 73.89, 74.638, 150.413]
  MoveL 198 to (-197.85, 348.32, -3.66) mm, rotated rx 174.1 ry -29.55 rz 11.83 deg; joints [2.654, -32.318, 122.84, -144.922, 73.887, 74.631, 150.404]
  MoveL 199 to (-197.85, 347.98, -3.31) mm, rotated rx 174.09 ry -29.55 rz 11.86 deg; joints [2.67, -32.335, 122.848, -144.908, 73.882, 74.615, 150.379]
  MoveL 200 to (-197.85, 347.5, -3.19) mm, rotated rx 174.07 ry -29.55 rz 11.9 deg; joints [2.675, -32.359, 122.862, -144.905, 73.877, 74.593, 150.345]
  MoveL 201 to (-197.85, 346.23, -3.19) mm, rotated rx 174.02 ry -29.54 rz 12 deg; joints [2.673, -32.423, 122.899, -144.914, 73.865, 74.536, 150.255]
  MoveL 202 to (-197.85, 345.75, -3.31) mm, rotated rx 174 ry -29.53 rz 12.04 deg; joints [2.667, -32.448, 122.914, -144.923, 73.861, 74.515, 150.221]
  MoveL 203 to (-197.85, 345.4, -3.66) mm, rotated rx 173.99 ry -29.53 rz 12.07 deg; joints [2.65, -32.466, 122.927, -144.943, 73.859, 74.5, 150.196]
  MoveL 204 to (-197.85, 345.28, -4.14) mm, rotated rx 173.98 ry -29.53 rz 12.08 deg; joints [2.627, -32.473, 122.933, -144.966, 73.86, 74.495, 150.187]
  MoveL 205 to (-197.85, 345.28, -8.4) mm, rotated rx 173.98 ry -29.53 rz 12.08 deg; joints [2.425, -32.477, 122.956, -145.171, 73.876, 74.505, 150.187]
  MoveL 206 to (-199.91, 345.28, -8.41) mm, rotated rx 173.84 ry -29.5 rz 12.37 deg; joints [2.419, -32.36, 122.938, -145.226, 73.984, 74.446, 149.93]
  MoveL 207 to (-206.05, 345.28, -11.57) mm, rotated rx 173.41 ry -29.42 rz 13.24 deg; joints [2.253, -32.015, 122.898, -145.543, 74.315, 74.279, 149.173]
  MoveL 208 to (-201.08, 345.28, -20.25) mm, rotated rx 173.75 ry -29.49 rz 12.54 deg; joints [1.854, -32.304, 122.984, -145.826, 74.087, 74.435, 149.785]
  MoveL 209 to (-201.08, 342.1, -20.25) mm, rotated rx 173.62 ry -29.46 rz 12.8 deg; joints [1.849, -32.464, 123.08, -145.852, 74.058, 74.292, 149.554]
  MoveL 210 to (-206.05, 342.1, -11.57) mm, rotated rx 173.28 ry -29.39 rz 13.5 deg; joints [2.248, -32.174, 122.995, -145.571, 74.288, 74.137, 148.939]
  MoveL 211 to (-199.87, 342.1, -8.41) mm, rotated rx 173.71 ry -29.48 rz 12.63 deg; joints [2.415, -32.522, 123.033, -145.25, 73.953, 74.304, 149.705]
  MoveL 212 to (-197.85, 342.1, -8.4) mm, rotated rx 173.85 ry -29.51 rz 12.34 deg; joints [2.42, -32.637, 123.051, -145.195, 73.847, 74.361, 149.958]
  MoveL 213 to (-197.85, 342.1, -4.14) mm, rotated rx 173.85 ry -29.51 rz 12.34 deg; joints [2.622, -32.633, 123.028, -144.99, 73.831, 74.351, 149.958]
  Set speed (38.1 mm/s)
  MoveL 214 to (-197.89, 342.1, -3.98) mm, rotated rx 173.85 ry -29.5 rz 12.34 deg; joints [2.63, -32.63, 123.026, -144.983, 73.832, 74.35, 149.953]
  MoveL 215 to (-198.05, 341.78, -3.7) mm, rotated rx 173.82 ry -29.5 rz 12.39 deg; joints [2.642, -32.637, 123.033, -144.977, 73.837, 74.33, 149.91]
  Set speed (76.2 mm/s)
  MoveL 216 to (-198.05, 339.25, -3.7) mm, rotated rx 173.72 ry -29.48 rz 12.61 deg; joints [2.638, -32.764, 123.109, -144.997, 73.813, 74.215, 149.724]
  Set speed (38.1 mm/s)
  MoveL 217 to (-197.89, 338.93, -3.98) mm, rotated rx 173.72 ry -29.48 rz 12.61 deg; joints [2.625, -32.789, 123.121, -145.008, 73.803, 74.205, 149.721]
  MoveL 218 to (-197.85, 338.93, -4.14) mm, rotated rx 173.72 ry -29.48 rz 12.6 deg; joints [2.618, -32.792, 123.122, -145.015, 73.802, 74.207, 149.726]
  Set speed (76.2 mm/s)
  MoveL 219 to (-197.85, 338.93, -8.4) mm, rotated rx 173.72 ry -29.48 rz 12.6 deg; joints [2.415, -32.796, 123.145, -145.22, 73.818, 74.217, 149.726]
  MoveL 220 to (-200.2, 338.93, -8.41) mm, rotated rx 173.55 ry -29.45 rz 12.94 deg; joints [2.409, -32.662, 123.125, -145.285, 73.942, 74.15, 149.43]
  MoveL 221 to (-206.05, 338.93, -11.57) mm, rotated rx 173.15 ry -29.36 rz 13.77 deg; joints [2.243, -32.331, 123.091, -145.6, 74.262, 73.994, 148.703]
  MoveL 222 to (-201.08, 338.93, -20.25) mm, rotated rx 173.49 ry -29.43 rz 13.07 deg; joints [1.844, -32.622, 123.175, -145.878, 74.03, 74.149, 149.32]
  MoveL 223 to (-201.08, 335.75, -20.25) mm, rotated rx 173.36 ry -29.41 rz 13.34 deg; joints [1.838, -32.78, 123.27, -145.906, 74.002, 74.005, 149.083]
  MoveL 224 to (-206.05, 335.75, -11.57) mm, rotated rx 173.01 ry -29.33 rz 14.04 deg; joints [2.237, -32.488, 123.187, -145.631, 74.236, 73.851, 148.463]
  MoveL 225 to (-200.15, 335.75, -8.41) mm, rotated rx 173.43 ry -29.42 rz 13.2 deg; joints [2.404, -32.823, 123.221, -145.311, 73.912, 74.007, 149.199]
  MoveL 226 to (-197.85, 335.75, -8.4) mm, rotated rx 173.59 ry -29.45 rz 12.87 deg; joints [2.41, -32.955, 123.239, -145.246, 73.789, 74.072, 149.491]
  MoveL 227 to (-197.85, 335.75, -4.14) mm, rotated rx 173.59 ry -29.45 rz 12.87 deg; joints [2.613, -32.951, 123.217, -145.041, 73.773, 74.062, 149.491]
  Set speed (38.1 mm/s)
  MoveL 228 to (-197.89, 335.75, -3.98) mm, rotated rx 173.59 ry -29.45 rz 12.88 deg; joints [2.62, -32.948, 123.215, -145.034, 73.775, 74.06, 149.485]
  MoveL 229 to (-198.05, 335.44, -3.7) mm, rotated rx 173.56 ry -29.45 rz 12.93 deg; joints [2.632, -32.955, 123.222, -145.028, 73.78, 74.04, 149.442]
  Set speed (76.2 mm/s)
  MoveL 230 to (-198.05, 332.9, -3.7) mm, rotated rx 173.45 ry -29.43 rz 13.15 deg; joints [2.628, -33.081, 123.298, -145.05, 73.758, 73.924, 149.251]
  Set speed (38.1 mm/s)
  MoveL 231 to (-197.89, 332.58, -3.98) mm, rotated rx 173.45 ry -29.43 rz 13.15 deg; joints [2.615, -33.106, 123.31, -145.061, 73.747, 73.914, 149.247]
  MoveL 232 to (-197.85, 332.58, -4.14) mm, rotated rx 173.45 ry -29.43 rz 13.14 deg; joints [2.608, -33.109, 123.311, -145.068, 73.746, 73.916, 149.252]
  Set speed (76.2 mm/s)
  MoveL 233 to (-197.85, 332.58, -8.4) mm, rotated rx 173.45 ry -29.43 rz 13.14 deg; joints [2.405, -33.113, 123.334, -145.273, 73.761, 73.926, 149.252]
  MoveL 234 to (-200.15, 332.58, -8.41) mm, rotated rx 173.29 ry -29.39 rz 13.48 deg; joints [2.398, -32.98, 123.316, -145.34, 73.885, 73.861, 148.96]
  MoveL 235 to (-206.05, 332.58, -11.57) mm, rotated rx 172.88 ry -29.3 rz 14.32 deg; joints [2.231, -32.644, 123.283, -145.662, 74.211, 73.706, 148.22]
  MoveL 236 to (-201.08, 332.58, -20.25) mm, rotated rx 173.23 ry -29.38 rz 13.61 deg; joints [1.833, -32.937, 123.365, -145.936, 73.975, 73.86, 148.843]
  MoveL 237 to (-201.08, 329.4, -20.25) mm, rotated rx 173.09 ry -29.35 rz 13.89 deg; joints [1.827, -33.094, 123.46, -145.967, 73.949, 73.714, 148.599]
  MoveL 238 to (-206.05, 329.4, -11.57) mm, rotated rx 172.74 ry -29.27 rz 14.6 deg; joints [2.225, -32.799, 123.38, -145.696, 74.186, 73.561, 147.973]
  MoveL 239 to (-200.15, 329.4, -8.41) mm, rotated rx 173.15 ry -29.36 rz 13.76 deg; joints [2.393, -33.137, 123.41, -145.37, 73.859, 73.715, 148.716]
  MoveL 240 to (-197.85, 329.4, -8.4) mm, rotated rx 173.32 ry -29.4 rz 13.42 deg; joints [2.4, -33.27, 123.428, -145.302, 73.734, 73.779, 149.01]
  MoveL 241 to (-197.85, 329.4, -4.14) mm, rotated rx 173.32 ry -29.4 rz 13.42 deg; joints [2.602, -33.266, 123.406, -145.096, 73.719, 73.769, 149.01]
  Set speed (38.1 mm/s)
  MoveL 242 to (-197.89, 329.4, -3.98) mm, rotated rx 173.32 ry -29.4 rz 13.43 deg; joints [2.61, -33.263, 123.404, -145.09, 73.72, 73.767, 149.005]
  MoveL 243 to (-198.05, 329.09, -3.7) mm, rotated rx 173.29 ry -29.39 rz 13.48 deg; joints [2.622, -33.27, 123.411, -145.084, 73.725, 73.747, 148.96]
  Set speed (76.2 mm/s)
  MoveL 244 to (-198.05, 326.55, -3.7) mm, rotated rx 173.18 ry -29.37 rz 13.7 deg; joints [2.617, -33.395, 123.487, -145.108, 73.704, 73.629, 148.764]
  Set speed (38.1 mm/s)
  MoveL 245 to (-197.89, 326.23, -3.98) mm, rotated rx 173.18 ry -29.37 rz 13.71 deg; joints [2.604, -33.42, 123.499, -145.12, 73.694, 73.619, 148.759]
  MoveL 246 to (-197.85, 326.23, -4.14) mm, rotated rx 173.18 ry -29.37 rz 13.7 deg; joints [2.597, -33.422, 123.5, -145.126, 73.692, 73.621, 148.765]
  Set speed (76.2 mm/s)
  MoveL 247 to (-197.85, 326.23, -8.4) mm, rotated rx 173.18 ry -29.37 rz 13.7 deg; joints [2.394, -33.427, 123.523, -145.332, 73.708, 73.632, 148.765]
  MoveL 248 to (-200.15, 326.23, -8.41) mm, rotated rx 173.02 ry -29.33 rz 14.04 deg; joints [2.387, -33.293, 123.505, -145.401, 73.833, 73.568, 148.469]
  MoveL 249 to (-206.05, 326.23, -11.57) mm, rotated rx 172.6 ry -29.24 rz 14.89 deg; joints [2.219, -32.953, 123.476, -145.73, 74.163, 73.415, 147.723]
  MoveL 250 to (-201.08, 326.23, -20.25) mm, rotated rx 172.95 ry -29.32 rz 14.17 deg; joints [1.821, -33.25, 123.555, -145.999, 73.923, 73.567, 148.352]
  MoveL 251 to (-201.08, 323.05, -20.25) mm, rotated rx 172.81 ry -29.29 rz 14.46 deg; joints [1.814, -33.405, 123.65, -146.033, 73.898, 73.42, 148.101]
  MoveL 252 to (-206.05, 323.05, -11.57) mm, rotated rx 172.46 ry -29.21 rz 15.17 deg; joints [2.212, -33.107, 123.572, -145.767, 74.14, 73.268, 147.47]
  MoveL 253 to (-200.15, 323.05, -8.41) mm, rotated rx 172.88 ry -29.3 rz 14.32 deg; joints [2.381, -33.448, 123.6, -145.434, 73.808, 73.42, 148.219]
  MoveL 254 to (-197.85, 323.05, -8.4) mm, rotated rx 173.04 ry -29.34 rz 13.98 deg; joints [2.388, -33.582, 123.617, -145.363, 73.682, 73.483, 148.516]
  MoveL 255 to (-197.85, 323.05, -4.14) mm, rotated rx 173.04 ry -29.34 rz 13.98 deg; joints [2.591, -33.578, 123.594, -145.158, 73.667, 73.472, 148.516]
  Set speed (38.1 mm/s)
  MoveL 256 to (-197.89, 323.05, -3.98) mm, rotated rx 173.04 ry -29.34 rz 13.99 deg; joints [2.598, -33.576, 123.593, -145.151, 73.669, 73.471, 148.51]
  MoveL 257 to (-198.05, 322.74, -3.7) mm, rotated rx 173.01 ry -29.33 rz 14.04 deg; joints [2.61, -33.582, 123.6, -145.146, 73.674, 73.451, 148.465]
  Set speed (76.2 mm/s)
  MoveL 258 to (-198.05, 320.2, -3.7) mm, rotated rx 172.9 ry -29.31 rz 14.27 deg; joints [2.606, -33.706, 123.676, -145.172, 73.654, 73.331, 148.262]
  Set speed (38.1 mm/s)
  MoveL 259 to (-197.89, 319.88, -3.98) mm, rotated rx 172.9 ry -29.31 rz 14.28 deg; joints [2.592, -33.731, 123.688, -145.184, 73.644, 73.322, 148.258]
  MoveL 260 to (-197.85, 319.88, -4.14) mm, rotated rx 172.9 ry -29.31 rz 14.27 deg; joints [2.585, -33.733, 123.689, -145.191, 73.642, 73.323, 148.263]
  Set speed (76.2 mm/s)
  MoveL 261 to (-197.85, 319.88, -8.4) mm, rotated rx 172.9 ry -29.31 rz 14.27 deg; joints [2.382, -33.738, 123.711, -145.396, 73.657, 73.334, 148.263]
  MoveL 262 to (-200.15, 319.88, -8.41) mm, rotated rx 172.74 ry -29.27 rz 14.61 deg; joints [2.375, -33.603, 123.695, -145.468, 73.784, 73.271, 147.965]
  MoveL 263 to (-206.05, 319.88, -11.57) mm, rotated rx 172.32 ry -29.17 rz 15.47 deg; joints [2.205, -33.26, 123.669, -145.804, 74.117, 73.12, 147.213]
  MoveL 264 to (-201.08, 319.88, -20.25) mm, rotated rx 172.67 ry -29.26 rz 14.75 deg; joints [1.808, -33.559, 123.745, -146.068, 73.874, 73.272, 147.846]
  MoveL 265 to (-201.08, 316.7, -20.25) mm, rotated rx 172.53 ry -29.22 rz 15.04 deg; joints [1.801, -33.713, 123.841, -146.104, 73.85, 73.122, 147.588]
  MoveL 266 to (-206.05, 316.7, -11.57) mm, rotated rx 172.17 ry -29.14 rz 15.76 deg; joints [2.198, -33.413, 123.765, -145.844, 74.096, 72.972, 146.952]
  MoveL 267 to (-200.15, 316.7, -8.41) mm, rotated rx 172.59 ry -29.24 rz 14.9 deg; joints [2.368, -33.757, 123.79, -145.504, 73.76, 73.121, 147.708]
  MoveL 268 to (-197.85, 316.7, -8.4) mm, rotated rx 172.76 ry -29.28 rz 14.56 deg; joints [2.376, -33.892, 123.806, -145.431, 73.633, 73.184, 148.007]
  MoveL 269 to (-197.85, 316.7, -4.14) mm, rotated rx 172.76 ry -29.28 rz 14.56 deg; joints [2.579, -33.888, 123.783, -145.225, 73.618, 73.173, 148.007]
  Set speed (38.1 mm/s)
  MoveL 270 to (-197.89, 316.7, -3.98) mm, rotated rx 172.76 ry -29.28 rz 14.57 deg; joints [2.586, -33.885, 123.782, -145.219, 73.62, 73.171, 148.001]
  MoveL 271 to (-198.05, 316.39, -3.7) mm, rotated rx 172.73 ry -29.27 rz 14.62 deg; joints [2.598, -33.891, 123.789, -145.214, 73.625, 73.151, 147.955]
  Set speed (76.2 mm/s)
  MoveL 272 to (-198.05, 313.85, -3.7) mm, rotated rx 172.61 ry -29.24 rz 14.86 deg; joints [2.593, -34.014, 123.865, -145.243, 73.606, 73.03, 147.747]
  Set speed (38.1 mm/s)
  MoveL 273 to (-197.89, 313.53, -3.98) mm, rotated rx 172.61 ry -29.24 rz 14.86 deg; joints [2.58, -34.039, 123.877, -145.255, 73.596, 73.02, 147.741]
  MoveL 274 to (-197.85, 313.53, -4.14) mm, rotated rx 172.62 ry -29.24 rz 14.86 deg; joints [2.572, -34.041, 123.878, -145.261, 73.594, 73.022, 147.747]
  Set speed (76.2 mm/s)
  MoveL 275 to (-197.85, 313.53, -8.4) mm, rotated rx 172.62 ry -29.24 rz 14.86 deg; joints [2.369, -34.045, 123.9, -145.467, 73.609, 73.033, 147.747]
  MoveL 276 to (-200.15, 313.53, -8.41) mm, rotated rx 172.45 ry -29.21 rz 15.2 deg; joints [2.361, -33.91, 123.885, -145.541, 73.738, 72.971, 147.446]
  MoveL 277 to (-206.05, 313.53, -11.57) mm, rotated rx 172.03 ry -29.1 rz 16.06 deg; joints [2.191, -33.564, 123.862, -145.885, 74.075, 72.823, 146.687]
  MoveL 278 to (-201.08, 313.53, -20.25) mm, rotated rx 172.38 ry -29.19 rz 15.34 deg; joints [1.794, -33.866, 123.936, -146.143, 73.827, 72.973, 147.327]
  MoveL 279 to (-201.08, 310.35, -20.25) mm, rotated rx 172.24 ry -29.15 rz 15.64 deg; joints [1.787, -34.018, 124.031, -146.183, 73.805, 72.822, 147.061]
  MoveL 280 to (-206.05, 310.35, -11.57) mm, rotated rx 171.88 ry -29.07 rz 16.36 deg; joints [2.183, -33.715, 123.958, -145.927, 74.055, 72.673, 146.419]
  MoveL 281 to (-200.15, 310.35, -8.41) mm, rotated rx 172.3 ry -29.17 rz 15.5 deg; joints [2.355, -34.062, 123.981, -145.58, 73.716, 72.82, 147.181]
  MoveL 282 to (-197.85, 310.35, -8.4) mm, rotated rx 172.47 ry -29.21 rz 15.16 deg; joints [2.363, -34.198, 123.995, -145.505, 73.586, 72.882, 147.483]
  MoveL 283 to (-197.85, 310.35, -4.14) mm, rotated rx 172.47 ry -29.21 rz 15.16 deg; joints [2.566, -34.194, 123.972, -145.299, 73.572, 72.87, 147.483]
  Set speed (38.1 mm/s)
  MoveL 284 to (-197.89, 310.35, -3.98) mm, rotated rx 172.47 ry -29.21 rz 15.16 deg; joints [2.573, -34.191, 123.971, -145.292, 73.574, 72.869, 147.478]
  MoveL 285 to (-198.05, 310.04, -3.7) mm, rotated rx 172.44 ry -29.2 rz 15.22 deg; joints [2.585, -34.197, 123.978, -145.288, 73.579, 72.848, 147.43]
  Set speed (76.2 mm/s)
  MoveL 286 to (-198.05, 307.5, -3.7) mm, rotated rx 172.32 ry -29.17 rz 15.46 deg; joints [2.579, -34.318, 124.054, -145.319, 73.562, 72.726, 147.216]
  Set speed (38.1 mm/s)
  MoveL 287 to (-197.89, 307.18, -3.98) mm, rotated rx 172.32 ry -29.17 rz 15.47 deg; joints [2.566, -34.343, 124.066, -145.331, 73.552, 72.716, 147.21]
  MoveL 288 to (-197.85, 307.18, -4.14) mm, rotated rx 172.32 ry -29.17 rz 15.46 deg; joints [2.559, -34.346, 124.067, -145.338, 73.55, 72.718, 147.216]
  Set speed (76.2 mm/s)
  MoveL 289 to (-197.85, 307.18, -8.4) mm, rotated rx 172.32 ry -29.17 rz 15.46 deg; joints [2.356, -34.35, 124.09, -145.544, 73.564, 72.729, 147.216]
  MoveL 290 to (-200.15, 307.18, -8.41) mm, rotated rx 172.15 ry -29.13 rz 15.81 deg; joints [2.347, -34.213, 124.076, -145.621, 73.695, 72.668, 146.912]
  MoveL 291 to (-206.05, 307.18, -11.57) mm, rotated rx 171.73 ry -29.03 rz 16.67 deg; joints [2.175, -33.865, 124.055, -145.972, 74.036, 72.522, 146.147]
  MoveL 292 to (-201.08, 307.18, -20.25) mm, rotated rx 172.09 ry -29.12 rz 15.94 deg; joints [1.779, -34.169, 124.127, -146.224, 73.784, 72.671, 146.792]
  MoveL 293 to (-201.08, 304.01, -20.25) mm, rotated rx 171.94 ry -29.08 rz 16.25 deg; joints [1.771, -34.319, 124.222, -146.268, 73.764, 72.518, 146.518]
  MoveL 294 to (-206.05, 304.01, -11.57) mm, rotated rx 171.58 ry -28.99 rz 16.98 deg; joints [2.167, -34.014, 124.152, -146.018, 74.017, 72.371, 145.871]
  MoveL 295 to (-200.15, 304.01, -8.41) mm, rotated rx 172 ry -29.1 rz 16.12 deg; joints [2.34, -34.364, 124.172, -145.664, 73.674, 72.515, 146.64]
  MoveL 296 to (-197.85, 304.01, -8.4) mm, rotated rx 172.17 ry -29.14 rz 15.77 deg; joints [2.348, -34.502, 124.185, -145.585, 73.543, 72.576, 146.944]
  MoveL 297 to (-197.85, 304.01, -4.14) mm, rotated rx 172.17 ry -29.14 rz 15.77 deg; joints [2.551, -34.497, 124.162, -145.379, 73.529, 72.564, 146.944]
  Set speed (38.1 mm/s)
  MoveL 298 to (-197.89, 304.01, -3.98) mm, rotated rx 172.17 ry -29.14 rz 15.78 deg; joints [2.559, -34.494, 124.161, -145.373, 73.531, 72.563, 146.938]
  MoveL 299 to (-198.05, 303.69, -3.7) mm, rotated rx 172.14 ry -29.13 rz 15.83 deg; joints [2.571, -34.5, 124.168, -145.369, 73.537, 72.542, 146.89]
  Set speed (76.2 mm/s)
  MoveL 300 to (-198.05, 301.15, -3.7) mm, rotated rx 172.02 ry -29.1 rz 16.08 deg; joints [2.565, -34.62, 124.244, -145.403, 73.521, 72.419, 146.669]
  Set speed (38.1 mm/s)
  MoveL 301 to (-197.89, 300.83, -3.98) mm, rotated rx 172.02 ry -29.1 rz 16.09 deg; joints [2.551, -34.645, 124.256, -145.415, 73.511, 72.409, 146.663]
  MoveL 302 to (-197.85, 300.83, -4.14) mm, rotated rx 172.02 ry -29.1 rz 16.08 deg; joints [2.544, -34.648, 124.257, -145.422, 73.509, 72.41, 146.669]
  Set speed (76.2 mm/s)
  MoveL 303 to (-197.85, 300.83, -8.4) mm, rotated rx 172.02 ry -29.1 rz 16.08 deg; joints [2.341, -34.652, 124.28, -145.628, 73.523, 72.422, 146.669]
  MoveL 304 to (-200.15, 300.83, -8.41) mm, rotated rx 171.85 ry -29.06 rz 16.43 deg; joints [2.332, -34.514, 124.267, -145.708, 73.655, 72.361, 146.363]
  MoveL 305 to (-206.05, 300.83, -11.57) mm, rotated rx 171.43 ry -28.95 rz 17.3 deg; joints [2.159, -34.163, 124.249, -146.066, 74, 72.219, 145.591]
  MoveL 306 to (-201.08, 300.83, -20.25) mm, rotated rx 171.78 ry -29.04 rz 16.57 deg; joints [1.763, -34.469, 124.318, -146.313, 73.744, 72.365, 146.241]
  MoveL 307 to (-201.08, 297.66, -20.25) mm, rotated rx 171.63 ry -29 rz 16.89 deg; joints [1.755, -34.618, 124.414, -146.36, 73.725, 72.212, 145.96]
  MoveL 308 to (-206.05, 297.66, -11.57) mm, rotated rx 171.27 ry -28.9 rz 17.62 deg; joints [2.15, -34.31, 124.347, -146.116, 73.983, 72.066, 145.308]
  MoveL 309 to (-200.15, 297.66, -8.41) mm, rotated rx 171.7 ry -29.02 rz 16.75 deg; joints [2.324, -34.663, 124.363, -145.754, 73.636, 72.207, 146.082]
  MoveL 310 to (-197.85, 297.66, -8.4) mm, rotated rx 171.86 ry -29.06 rz 16.4 deg; joints [2.333, -34.802, 124.375, -145.673, 73.504, 72.267, 146.389]
  MoveL 311 to (-197.85, 297.66, -4.14) mm, rotated rx 171.86 ry -29.06 rz 16.4 deg; joints [2.536, -34.797, 124.353, -145.466, 73.49, 72.255, 146.389]
  Set speed (38.1 mm/s)
  MoveL 312 to (-197.89, 297.66, -3.98) mm, rotated rx 171.86 ry -29.06 rz 16.41 deg; joints [2.544, -34.794, 124.352, -145.46, 73.492, 72.254, 146.383]
  MoveL 313 to (-198.05, 297.34, -3.7) mm, rotated rx 171.83 ry -29.05 rz 16.46 deg; joints [2.555, -34.8, 124.359, -145.457, 73.498, 72.233, 146.334]
  Set speed (76.2 mm/s)
  MoveL 314 to (-198.05, 294.8, -3.7) mm, rotated rx 171.71 ry -29.02 rz 16.72 deg; joints [2.549, -34.919, 124.435, -145.494, 73.483, 72.109, 146.107]
  Set speed (38.1 mm/s)
  MoveL 315 to (-197.89, 294.48, -3.98) mm, rotated rx 171.71 ry -29.02 rz 16.73 deg; joints [2.536, -34.943, 124.447, -145.507, 73.473, 72.098, 146.099]
  MoveL 316 to (-197.85, 294.48, -4.14) mm, rotated rx 171.71 ry -29.02 rz 16.72 deg; joints [2.528, -34.946, 124.448, -145.513, 73.471, 72.099, 146.105]
  Set speed (76.2 mm/s)
  MoveL 317 to (-197.85, 294.48, -8.4) mm, rotated rx 171.71 ry -29.02 rz 16.72 deg; joints [2.325, -34.95, 124.47, -145.72, 73.485, 72.111, 146.105]
  MoveL 318 to (-200.15, 294.48, -8.41) mm, rotated rx 171.54 ry -28.98 rz 17.07 deg; joints [2.315, -34.811, 124.459, -145.802, 73.618, 72.052, 145.797]
  MoveL 319 to (-206.05, 294.48, -11.57) mm, rotated rx 171.11 ry -28.86 rz 17.95 deg; joints [2.141, -34.457, 124.444, -146.168, 73.967, 71.912, 145.019]
  MoveL 320 to (-201.08, 294.48, -20.25) mm, rotated rx 171.47 ry -28.96 rz 17.21 deg; joints [1.746, -34.766, 124.51, -146.409, 73.707, 72.057, 145.674]
  MoveL 321 to (-201.08, 291.31, -20.25) mm, rotated rx 171.31 ry -28.91 rz 17.54 deg; joints [1.737, -34.913, 124.607, -146.46, 73.69, 71.902, 145.384]
  MoveL 322 to (-206.05, 291.31, -11.57) mm, rotated rx 170.96 ry -28.81 rz 18.28 deg; joints [2.132, -34.603, 124.542, -146.221, 73.952, 71.758, 144.727]
  MoveL 323 to (-200.15, 291.31, -8.41) mm, rotated rx 171.38 ry -28.93 rz 17.4 deg; joints [2.307, -34.958, 124.556, -145.852, 73.602, 71.896, 145.508]
  MoveL 324 to (-197.85, 291.31, -8.4) mm, rotated rx 171.55 ry -28.98 rz 17.05 deg; joints [2.316, -35.098, 124.566, -145.768, 73.468, 71.955, 145.817]
  MoveL 325 to (-197.85, 291.31, -4.14) mm, rotated rx 171.55 ry -28.98 rz 17.05 deg; joints [2.52, -35.094, 124.544, -145.561, 73.454, 71.943, 145.817]
  Set speed (38.1 mm/s)
  MoveL 326 to (-197.89, 291.31, -3.98) mm, rotated rx 171.55 ry -28.98 rz 17.05 deg; joints [2.527, -35.091, 124.543, -145.555, 73.456, 71.941, 145.811]
  MoveL 327 to (-198.05, 290.99, -3.7) mm, rotated rx 171.52 ry -28.97 rz 17.11 deg; joints [2.539, -35.096, 124.55, -145.553, 73.462, 71.921, 145.761]
  Set speed (76.2 mm/s)
  MoveL 328 to (-198.05, 288.45, -3.7) mm, rotated rx 171.39 ry -28.94 rz 17.37 deg; joints [2.532, -35.214, 124.627, -145.593, 73.449, 71.795, 145.527]
  Set speed (38.1 mm/s)
  MoveL 329 to (-197.89, 288.13, -3.98) mm, rotated rx 171.39 ry -28.93 rz 17.38 deg; joints [2.518, -35.238, 124.639, -145.606, 73.439, 71.784, 145.519]
  MoveL 330 to (-197.85, 288.13, -4.14) mm, rotated rx 171.39 ry -28.94 rz 17.38 deg; joints [2.511, -35.241, 124.64, -145.612, 73.437, 71.786, 145.525]
  Set speed (76.2 mm/s)
  MoveL 331 to (-197.85, 288.13, -8.4) mm, rotated rx 171.39 ry -28.94 rz 17.38 deg; joints [2.307, -35.246, 124.662, -145.819, 73.451, 71.798, 145.525]
  MoveL 332 to (-200.15, 288.13, -8.41) mm, rotated rx 171.22 ry -28.89 rz 17.73 deg; joints [2.298, -35.105, 124.652, -145.905, 73.586, 71.74, 145.214]
  MoveL 333 to (-206.05, 288.13, -11.57) mm, rotated rx 170.8 ry -28.77 rz 18.61 deg; joints [2.122, -34.748, 124.64, -146.277, 73.938, 71.602, 144.431]
  MoveL 334 to (-201.08, 288.13, -20.25) mm, rotated rx 171.15 ry -28.87 rz 17.87 deg; joints [1.728, -35.06, 124.704, -146.513, 73.674, 71.746, 145.09]
  MoveL 335 to (-201.08, 284.96, -20.25) mm, rotated rx 170.99 ry -28.82 rz 18.2 deg; joints [1.718, -35.205, 124.801, -146.568, 73.659, 71.589, 144.792]
  MoveL 336 to (-206.05, 284.96, -11.57) mm, rotated rx 170.63 ry -28.72 rz 18.95 deg; joints [2.112, -34.893, 124.739, -146.335, 73.925, 71.447, 144.13]
  MoveL 337 to (-200.15, 284.96, -8.41) mm, rotated rx 171.06 ry -28.84 rz 18.06 deg; joints [2.288, -35.251, 124.749, -145.959, 73.571, 71.582, 144.916]
  MoveL 338 to (-197.85, 284.96, -8.4) mm, rotated rx 171.23 ry -28.89 rz 17.71 deg; joints [2.298, -35.392, 124.759, -145.872, 73.435, 71.64, 145.228]
  MoveL 339 to (-197.85, 284.96, -4.14) mm, rotated rx 171.23 ry -28.89 rz 17.71 deg; joints [2.502, -35.387, 124.736, -145.664, 73.422, 71.628, 145.228]
  Set speed (38.1 mm/s)
  MoveL 340 to (-197.89, 284.96, -3.98) mm, rotated rx 171.23 ry -28.89 rz 17.72 deg; joints [2.509, -35.385, 124.735, -145.658, 73.424, 71.626, 145.222]
  MoveL 341 to (-198.05, 284.64, -3.7) mm, rotated rx 171.2 ry -28.88 rz 17.78 deg; joints [2.521, -35.389, 124.743, -145.656, 73.431, 71.605, 145.17]
  Set speed (76.2 mm/s)
  MoveL 342 to (-198.05, 282.1, -3.7) mm, rotated rx 171.07 ry -28.84 rz 18.05 deg; joints [2.513, -35.506, 124.82, -145.7, 73.419, 71.479, 144.929]
  Set speed (38.1 mm/s)
  MoveL 343 to (-197.89, 281.78, -3.98) mm, rotated rx 171.06 ry -28.84 rz 18.06 deg; joints [2.5, -35.53, 124.832, -145.713, 73.409, 71.467, 144.921]
  MoveL 344 to (-197.85, 281.78, -4.14) mm, rotated rx 171.06 ry -28.84 rz 18.05 deg; joints [2.493, -35.533, 124.833, -145.719, 73.407, 71.469, 144.926]
  Set speed (76.2 mm/s)
  MoveL 345 to (-197.85, 281.78, -8.4) mm, rotated rx 171.06 ry -28.84 rz 18.05 deg; joints [2.289, -35.537, 124.855, -145.927, 73.42, 71.481, 144.926]
  MoveL 346 to (-200.15, 281.78, -8.41) mm, rotated rx 170.89 ry -28.79 rz 18.4 deg; joints [2.279, -35.396, 124.846, -146.015, 73.557, 71.424, 144.613]
  MoveL 347 to (-206.05, 281.78, -11.57) mm, rotated rx 170.47 ry -28.67 rz 19.29 deg; joints [2.101, -35.036, 124.838, -146.396, 73.912, 71.29, 143.824]
  MoveL 348 to (-201.08, 281.78, -20.25) mm, rotated rx 170.83 ry -28.78 rz 18.55 deg; joints [1.708, -35.35, 124.898, -146.626, 73.645, 71.431, 144.489]
  MoveL 349 to (-201.08, 278.61, -20.25) mm, rotated rx 170.66 ry -28.73 rz 18.89 deg; joints [1.698, -35.494, 124.996, -146.686, 73.632, 71.273, 144.181]
  MoveL 350 to (-206.05, 278.61, -11.57) mm, rotated rx 170.3 ry -28.62 rz 19.64 deg; joints [2.091, -35.179, 124.937, -146.458, 73.901, 71.133, 143.515]
  MoveL 351 to (-200.15, 278.61, -8.41) mm, rotated rx 170.73 ry -28.75 rz 18.75 deg; joints [2.269, -35.54, 124.944, -146.074, 73.543, 71.265, 144.306]
  MoveL 352 to (-197.85, 278.61, -8.4) mm, rotated rx 170.9 ry -28.8 rz 18.4 deg; joints [2.279, -35.682, 124.952, -145.984, 73.406, 71.322, 144.621]
  MoveL 353 to (-197.85, 278.61, -4.14) mm, rotated rx 170.9 ry -28.8 rz 18.4 deg; joints [2.483, -35.677, 124.93, -145.776, 73.393, 71.309, 144.621]
  Set speed (38.1 mm/s)
  MoveL 354 to (-197.89, 278.61, -3.98) mm, rotated rx 170.89 ry -28.8 rz 18.4 deg; joints [2.49, -35.675, 124.929, -145.77, 73.395, 71.308, 144.615]
  MoveL 355 to (-198.05, 278.29, -3.7) mm, rotated rx 170.87 ry -28.79 rz 18.46 deg; joints [2.502, -35.679, 124.937, -145.769, 73.402, 71.287, 144.562]
  Set speed (76.2 mm/s)
  MoveL 356 to (-198.05, 275.75, -3.7) mm, rotated rx 170.73 ry -28.75 rz 18.74 deg; joints [2.494, -35.794, 125.015, -145.816, 73.392, 71.159, 144.314]
  Set speed (38.1 mm/s)
  MoveL 357 to (-197.89, 275.43, -3.98) mm, rotated rx 170.73 ry -28.75 rz 18.75 deg; joints [2.48, -35.818, 125.026, -145.829, 73.382, 71.148, 144.304]
  MoveL 358 to (-197.85, 275.43, -4.14) mm, rotated rx 170.73 ry -28.75 rz 18.75 deg; joints [2.473, -35.821, 125.027, -145.836, 73.38, 71.149, 144.31]
  Set speed (76.2 mm/s)
  MoveL 359 to (-197.85, 275.43, -8.4) mm, rotated rx 170.73 ry -28.75 rz 18.75 deg; joints [2.269, -35.826, 125.049, -146.043, 73.393, 71.162, 144.31]
  MoveL 360 to (-200.15, 275.43, -8.41) mm, rotated rx 170.56 ry -28.7 rz 19.1 deg; joints [2.258, -35.683, 125.042, -146.135, 73.531, 71.106, 143.995]
  MoveL 361 to (-206.05, 275.43, -11.57) mm, rotated rx 170.13 ry -28.56 rz 19.99 deg; joints [2.079, -35.321, 125.036, -146.523, 73.89, 70.975, 143.2]
  MoveL 362 to (-201.08, 275.43, -20.25) mm, rotated rx 170.49 ry -28.67 rz 19.24 deg; joints [1.687, -35.637, 125.094, -146.748, 73.62, 71.114, 143.869]
  MoveL 363 to (-201.08, 272.26, -20.25) mm, rotated rx 170.32 ry -28.62 rz 19.6 deg; joints [1.675, -35.779, 125.192, -146.812, 73.609, 70.954, 143.552]
  MoveL 364 to (-206.05, 272.26, -11.57) mm, rotated rx 169.96 ry -28.51 rz 20.35 deg; joints [2.068, -35.462, 125.136, -146.591, 73.881, 70.816, 142.881]
  MoveL 365 to (-200.15, 272.26, -8.41) mm, rotated rx 170.39 ry -28.64 rz 19.46 deg; joints [2.247, -35.825, 125.14, -146.198, 73.52, 70.946, 143.678]
  MoveL 366 to (-197.85, 272.26, -8.4) mm, rotated rx 170.56 ry -28.7 rz 19.1 deg; joints [2.258, -35.968, 125.147, -146.105, 73.382, 71.001, 143.995]
  MoveL 367 to (-197.85, 272.26, -4.14) mm, rotated rx 170.56 ry -28.7 rz 19.1 deg; joints [2.462, -35.964, 125.125, -145.897, 73.369, 70.988, 143.995]
  Set speed (38.1 mm/s)
  MoveL 368 to (-197.89, 272.26, -3.98) mm, rotated rx 170.56 ry -28.69 rz 19.11 deg; joints [2.47, -35.961, 125.124, -145.891, 73.371, 70.987, 143.989]
  MoveL 369 to (-198.05, 271.94, -3.7) mm, rotated rx 170.53 ry -28.69 rz 19.17 deg; joints [2.481, -35.965, 125.132, -145.891, 73.378, 70.966, 143.935]
  Set speed (76.2 mm/s)
  MoveL 370 to (-198.05, 269.4, -3.7) mm, rotated rx 170.39 ry -28.64 rz 19.46 deg; joints [2.473, -36.079, 125.211, -145.942, 73.37, 70.837, 143.679]
  Set speed (38.1 mm/s)
  MoveL 371 to (-197.89, 269.08, -3.98) mm, rotated rx 170.38 ry -28.64 rz 19.47 deg; joints [2.459, -36.103, 125.223, -145.955, 73.36, 70.825, 143.669]
  MoveL 372 to (-197.85, 269.08, -4.14) mm, rotated rx 170.39 ry -28.64 rz 19.46 deg; joints [2.452, -36.106, 125.224, -145.961, 73.358, 70.827, 143.675]
  Set speed (76.2 mm/s)
  MoveL 373 to (-197.85, 269.08, -8.4) mm, rotated rx 170.39 ry -28.64 rz 19.46 deg; joints [2.247, -36.11, 125.245, -146.169, 73.371, 70.839, 143.675]
  MoveL 374 to (-200.15, 269.08, -8.41) mm, rotated rx 170.22 ry -28.59 rz 19.82 deg; joints [2.236, -35.967, 125.239, -146.264, 73.51, 70.785, 143.357]
  MoveL 375 to (-206.05, 269.08, -11.57) mm, rotated rx 169.79 ry -28.45 rz 20.71 deg; joints [2.056, -35.602, 125.237, -146.661, 73.873, 70.657, 142.557]
  MoveL 376 to (-201.08, 269.08, -20.25) mm, rotated rx 170.15 ry -28.57 rz 19.96 deg; joints [1.664, -35.92, 125.291, -146.879, 73.598, 70.794, 143.23]
  MoveL 377 to (-201.08, 265.91, -20.25) mm, rotated rx 169.97 ry -28.51 rz 20.33 deg; joints [1.652, -36.06, 125.391, -146.948, 73.589, 70.632, 142.904]
  MoveL 378 to (-206.05, 265.91, -11.57) mm, rotated rx 169.61 ry -28.39 rz 21.08 deg; joints [2.043, -35.741, 125.338, -146.733, 73.865, 70.497, 142.228]
  MoveL 379 to (-200.15, 265.91, -8.41) mm, rotated rx 170.04 ry -28.53 rz 20.18 deg; joints [2.225, -36.107, 125.339, -146.333, 73.501, 70.623, 143.031]
  MoveL 380 to (-197.85, 265.91, -8.4) mm, rotated rx 170.21 ry -28.59 rz 19.83 deg; joints [2.236, -36.252, 125.344, -146.236, 73.361, 70.677, 143.349]
  MoveL 381 to (-197.85, 265.91, -4.14) mm, rotated rx 170.21 ry -28.59 rz 19.83 deg; joints [2.44, -36.247, 125.322, -146.028, 73.348, 70.664, 143.349]
  Set speed (38.1 mm/s)
  MoveL 382 to (-197.89, 265.91, -3.98) mm, rotated rx 170.21 ry -28.59 rz 19.83 deg; joints [2.448, -36.244, 125.321, -146.022, 73.35, 70.663, 143.344]
  MoveL 383 to (-198.05, 265.59, -3.7) mm, rotated rx 170.18 ry -28.58 rz 19.89 deg; joints [2.459, -36.248, 125.33, -146.022, 73.358, 70.642, 143.289]
  Set speed (76.2 mm/s)
  MoveL 384 to (-198.05, 263.05, -3.7) mm, rotated rx 170.04 ry -28.53 rz 20.19 deg; joints [2.45, -36.36, 125.409, -146.078, 73.351, 70.512, 143.024]
  Set speed (38.1 mm/s)
  MoveL 385 to (-197.89, 262.73, -3.98) mm, rotated rx 170.03 ry -28.53 rz 20.2 deg; joints [2.436, -36.384, 125.421, -146.091, 73.342, 70.5, 143.013]
  MoveL 386 to (-197.85, 262.73, -4.14) mm, rotated rx 170.03 ry -28.53 rz 20.2 deg; joints [2.429, -36.387, 125.422, -146.097, 73.34, 70.501, 143.019]
  Set speed (76.2 mm/s)
  MoveL 387 to (-197.85, 262.73, -8.4) mm, rotated rx 170.03 ry -28.53 rz 20.2 deg; joints [2.224, -36.392, 125.443, -146.305, 73.352, 70.514, 143.019]
  MoveL 388 to (-200.15, 262.73, -8.41) mm, rotated rx 169.86 ry -28.47 rz 20.55 deg; joints [2.213, -36.247, 125.439, -146.404, 73.493, 70.461, 142.7]
  MoveL 389 to (-206.05, 262.73, -11.57) mm, rotated rx 169.44 ry -28.33 rz 21.45 deg; joints [2.031, -35.879, 125.439, -146.808, 73.859, 70.337, 141.895]
  MoveL 390 to (-201.08, 262.73, -20.25) mm, rotated rx 169.8 ry -28.45 rz 20.7 deg; joints [1.639, -36.2, 125.491, -147.02, 73.581, 70.471, 142.572]
  MoveL 391 to (-201.08, 259.56, -20.25) mm, rotated rx 169.62 ry -28.39 rz 21.07 deg; joints [1.626, -36.338, 125.591, -147.095, 73.574, 70.308, 142.235]
  MoveL 392 to (-206.05, 259.56, -11.57) mm, rotated rx 169.26 ry -28.27 rz 21.83 deg; joints [2.017, -36.016, 125.541, -146.886, 73.853, 70.175, 141.556]
  MoveL 393 to (-200.15, 259.56, -8.41) mm, rotated rx 169.68 ry -28.42 rz 20.93 deg; joints [2.2, -36.386, 125.539, -146.477, 73.486, 70.298, 142.363]
  MoveL 394 to (-197.85, 259.56, -8.4) mm, rotated rx 169.86 ry -28.47 rz 20.57 deg; joints [2.212, -36.531, 125.543, -146.377, 73.344, 70.351, 142.684]
  MoveL 395 to (-197.85, 259.56, -4.14) mm, rotated rx 169.86 ry -28.47 rz 20.57 deg; joints [2.417, -36.526, 125.521, -146.169, 73.332, 70.338, 142.684]
  Set speed (38.1 mm/s)
  MoveL 396 to (-197.89, 259.56, -3.98) mm, rotated rx 169.85 ry -28.47 rz 20.58 deg; joints [2.424, -36.524, 125.521, -146.163, 73.334, 70.336, 142.678]
  MoveL 397 to (-198.05, 259.24, -3.7) mm, rotated rx 169.82 ry -28.46 rz 20.64 deg; joints [2.435, -36.527, 125.529, -146.164, 73.342, 70.315, 142.622]
  Set speed (76.2 mm/s)
  MoveL 398 to (-198.05, 256.7, -3.7) mm, rotated rx 169.68 ry -28.41 rz 20.95 deg; joints [2.425, -36.638, 125.609, -146.224, 73.337, 70.184, 142.35]
  Set speed (38.1 mm/s)
  MoveL 399 to (-197.89, 256.38, -3.98) mm, rotated rx 169.67 ry -28.41 rz 20.96 deg; joints [2.412, -36.662, 125.621, -146.238, 73.328, 70.172, 142.338]
  MoveL 400 to (-197.85, 256.38, -4.14) mm, rotated rx 169.67 ry -28.41 rz 20.95 deg; joints [2.404, -36.665, 125.622, -146.244, 73.326, 70.173, 142.344]
  Set speed (76.2 mm/s)
  MoveL 401 to (-197.85, 256.38, -8.4) mm, rotated rx 169.67 ry -28.41 rz 20.95 deg; joints [2.199, -36.669, 125.643, -146.452, 73.338, 70.186, 142.344]
  MoveL 402 to (-200.15, 256.38, -8.41) mm, rotated rx 169.5 ry -28.35 rz 21.31 deg; joints [2.187, -36.523, 125.64, -146.554, 73.48, 70.134, 142.022]
  MoveL 403 to (-206.05, 256.38, -11.57) mm, rotated rx 169.08 ry -28.2 rz 22.22 deg; joints [2.004, -36.153, 125.644, -146.966, 73.849, 70.014, 141.212]
  MoveL 404 to (-201.08, 256.38, -20.25) mm, rotated rx 169.44 ry -28.33 rz 21.46 deg; joints [1.613, -36.476, 125.692, -147.172, 73.568, 70.145, 141.894]
  MoveL 405 to (-201.08, 253.21, -20.25) mm, rotated rx 169.25 ry -28.27 rz 21.84 deg; joints [1.599, -36.613, 125.794, -147.253, 73.563, 69.981, 141.546]
  MoveL 406 to (-206.05, 253.21, -11.57) mm, rotated rx 168.89 ry -28.14 rz 22.61 deg; joints [1.989, -36.289, 125.747, -147.05, 73.846, 69.851, 140.863]
  MoveL 407 to (-200.15, 253.21, -8.41) mm, rotated rx 169.32 ry -28.29 rz 21.7 deg; joints [2.174, -36.66, 125.742, -146.633, 73.475, 69.97, 141.675]
  MoveL 408 to (-197.85, 253.21, -8.4) mm, rotated rx 169.49 ry -28.35 rz 21.34 deg; joints [2.186, -36.807, 125.744, -146.53, 73.332, 70.021, 141.998]
  MoveL 409 to (-197.85, 253.21, -4.14) mm, rotated rx 169.49 ry -28.35 rz 21.34 deg; joints [2.391, -36.802, 125.723, -146.322, 73.32, 70.008, 141.998]
  Set speed (38.1 mm/s)
  MoveL 410 to (-197.89, 253.21, -3.98) mm, rotated rx 169.49 ry -28.35 rz 21.35 deg; joints [2.399, -36.799, 125.722, -146.316, 73.322, 70.007, 141.992]
  MoveL 411 to (-198.05, 252.89, -3.7) mm, rotated rx 169.46 ry -28.34 rz 21.41 deg; joints [2.41, -36.803, 125.731, -146.317, 73.331, 69.986, 141.934]
  Set speed (76.2 mm/s)
  MoveL 412 to (-198.05, 250.35, -3.7) mm, rotated rx 169.31 ry -28.29 rz 21.72 deg; joints [2.399, -36.912, 125.812, -146.382, 73.328, 69.853, 141.653]
  Set speed (38.1 mm/s)
  MoveL 413 to (-197.89, 250.03, -3.98) mm, rotated rx 169.3 ry -28.28 rz 21.74 deg; joints [2.385, -36.936, 125.824, -146.396, 73.318, 69.841, 141.64]
  MoveL 414 to (-197.85, 250.03, -4.14) mm, rotated rx 169.3 ry -28.28 rz 21.73 deg; joints [2.378, -36.939, 125.825, -146.402, 73.316, 69.842, 141.646]
  Set speed (76.2 mm/s)
  MoveL 415 to (-197.85, 250.03, -8.4) mm, rotated rx 169.3 ry -28.28 rz 21.73 deg; joints [2.173, -36.943, 125.846, -146.611, 73.328, 69.856, 141.646]
  MoveL 416 to (-200.15, 250.03, -8.41) mm, rotated rx 169.13 ry -28.22 rz 22.09 deg; joints [2.16, -36.796, 125.844, -146.715, 73.471, 69.805, 141.323]
  MoveL 417 to (-206.05, 250.03, -11.57) mm, rotated rx 168.71 ry -28.07 rz 23 deg; joints [1.975, -36.423, 125.851, -147.136, 73.843, 69.688, 140.509]
  MoveL 418 to (-201.08, 250.03, -20.25) mm, rotated rx 169.07 ry -28.2 rz 22.24 deg; joints [1.585, -36.748, 125.896, -147.336, 73.559, 69.817, 141.194]
  MoveL 419 to (-201.08, 246.86, -20.25) mm, rotated rx 168.88 ry -28.13 rz 22.64 deg; joints [1.57, -36.883, 125.999, -147.422, 73.557, 69.652, 140.836]
  MoveL 420 to (-206.05, 246.86, -11.57) mm, rotated rx 168.52 ry -28 rz 23.4 deg; joints [1.959, -36.557, 125.955, -147.226, 73.842, 69.525, 140.149]
  MoveL 421 to (-200.15, 246.86, -8.41) mm, rotated rx 168.95 ry -28.16 rz 22.49 deg; joints [2.145, -36.931, 125.947, -146.801, 73.469, 69.64, 140.965]
  MoveL 422 to (-197.85, 246.86, -8.4) mm, rotated rx 169.12 ry -28.22 rz 22.13 deg; joints [2.159, -37.079, 125.948, -146.694, 73.325, 69.689, 141.29]
  MoveL 423 to (-197.85, 246.86, -4.14) mm, rotated rx 169.12 ry -28.22 rz 22.13 deg; joints [2.364, -37.074, 125.927, -146.486, 73.313, 69.676, 141.29]
  Set speed (38.1 mm/s)
  MoveL 424 to (-197.89, 246.86, -3.98) mm, rotated rx 169.11 ry -28.22 rz 22.14 deg; joints [2.371, -37.071, 125.926, -146.48, 73.315, 69.675, 141.284]
  MoveL 425 to (-198.05, 246.54, -3.7) mm, rotated rx 169.08 ry -28.21 rz 22.2 deg; joints [2.382, -37.075, 125.935, -146.482, 73.324, 69.654, 141.225]
  Set speed (76.2 mm/s)
  MoveL 426 to (-198.05, 244, -3.7) mm, rotated rx 168.93 ry -28.15 rz 22.52 deg; joints [2.37, -37.182, 126.017, -146.552, 73.322, 69.52, 140.935]
  Set speed (38.1 mm/s)
  MoveL 427 to (-197.89, 243.69, -3.98) mm, rotated rx 168.92 ry -28.15 rz 22.54 deg; joints [2.357, -37.206, 126.029, -146.566, 73.313, 69.508, 140.921]
  MoveL 428 to (-197.85, 243.69, -4.14) mm, rotated rx 168.93 ry -28.15 rz 22.53 deg; joints [2.349, -37.209, 126.03, -146.572, 73.311, 69.509, 140.927]
  Set speed (76.2 mm/s)
  MoveL 429 to (-197.85, 243.69, -8.4) mm, rotated rx 168.93 ry -28.15 rz 22.53 deg; joints [2.144, -37.214, 126.051, -146.781, 73.323, 69.523, 140.927]
  MoveL 430 to (-200.15, 243.69, -8.41) mm, rotated rx 168.75 ry -28.09 rz 22.9 deg; joints [2.13, -37.066, 126.05, -146.889, 73.467, 69.473, 140.602]
  MoveL 431 to (-206.05, 243.69, -11.57) mm, rotated rx 168.33 ry -27.92 rz 23.8 deg; joints [1.944, -36.69, 126.06, -147.318, 73.842, 69.361, 139.784]
  MoveL 432 to (-201.08, 243.69, -20.25) mm, rotated rx 168.69 ry -28.06 rz 23.04 deg; joints [1.554, -37.017, 126.103, -147.512, 73.555, 69.486, 140.472]
  MoveL 433 to (-201.08, 240.51, -20.25) mm, rotated rx 168.49 ry -27.99 rz 23.45 deg; joints [1.538, -37.15, 126.207, -147.604, 73.555, 69.32, 140.103]
  MoveL 434 to (-206.05, 240.51, -11.57) mm, rotated rx 168.14 ry -27.85 rz 24.21 deg; joints [1.927, -36.822, 126.166, -147.414, 73.843, 69.196, 139.413]
  MoveL 435 to (-200.15, 240.51, -8.41) mm, rotated rx 168.56 ry -28.01 rz 23.31 deg; joints [2.115, -37.199, 126.155, -146.981, 73.467, 69.307, 140.233]
  MoveL 436 to (-197.85, 240.51, -8.4) mm, rotated rx 168.73 ry -28.08 rz 22.94 deg; joints [2.129, -37.347, 126.155, -146.871, 73.322, 69.355, 140.559]
  MoveL 437 to (-197.85, 240.51, -4.14) mm, rotated rx 168.73 ry -28.08 rz 22.94 deg; joints [2.334, -37.343, 126.134, -146.662, 73.31, 69.342, 140.559]
  Set speed (38.1 mm/s)
  MoveL 438 to (-197.89, 240.51, -3.98) mm, rotated rx 168.73 ry -28.08 rz 22.95 deg; joints [2.342, -37.34, 126.133, -146.656, 73.312, 69.34, 140.553]
  MoveL 439 to (-198.05, 240.19, -3.7) mm, rotated rx 168.7 ry -28.06 rz 23.02 deg; joints [2.352, -37.343, 126.142, -146.66, 73.322, 69.319, 140.493]
  Set speed (76.2 mm/s)
  MoveL 440 to (-198.05, 237.65, -3.7) mm, rotated rx 168.54 ry -28.01 rz 23.35 deg; joints [2.34, -37.449, 126.226, -146.734, 73.322, 69.185, 140.194]
  Set speed (38.1 mm/s)
  MoveL 441 to (-197.89, 237.34, -3.98) mm, rotated rx 168.53 ry -28 rz 23.37 deg; joints [2.326, -37.473, 126.238, -146.749, 73.313, 69.172, 140.179]
  MoveL 442 to (-197.85, 237.34, -4.14) mm, rotated rx 168.54 ry -28 rz 23.36 deg; joints [2.319, -37.475, 126.238, -146.755, 73.31, 69.174, 140.185]
  Set speed (76.2 mm/s)
  MoveL 443 to (-197.85, 237.34, -8.4) mm, rotated rx 168.54 ry -28 rz 23.36 deg; joints [2.113, -37.48, 126.26, -146.964, 73.322, 69.187, 140.185]
  MoveL 444 to (-200.15, 237.34, -8.41) mm, rotated rx 168.37 ry -27.94 rz 23.72 deg; joints [2.099, -37.331, 126.26, -147.076, 73.468, 69.14, 139.858]
  MoveL 445 to (-206.05, 237.34, -11.57) mm, rotated rx 167.94 ry -27.77 rz 24.63 deg; joints [1.91, -36.953, 126.273, -147.513, 73.845, 69.031, 139.036]
  MoveL 446 to (-201.08, 237.34, -20.25) mm, rotated rx 168.3 ry -27.91 rz 23.87 deg; joints [1.522, -37.282, 126.312, -147.701, 73.555, 69.153, 139.728]
  MoveL 447 to (-201.08, 234.16, -20.25) mm, rotated rx 168.1 ry -27.83 rz 24.29 deg; joints [1.505, -37.413, 126.418, -147.8, 73.557, 68.985, 139.347]
  MoveL 448 to (-206.05, 234.16, -11.57) mm, rotated rx 167.75 ry -27.69 rz 25.05 deg; joints [1.893, -37.083, 126.38, -147.616, 73.849, 68.865, 138.654]
  MoveL 449 to (-200.15, 234.16, -8.41) mm, rotated rx 168.17 ry -27.86 rz 24.14 deg; joints [2.082, -37.462, 126.366, -147.174, 73.47, 68.972, 139.477]
  MoveL 450 to (-197.85, 234.16, -8.4) mm, rotated rx 168.34 ry -27.93 rz 23.78 deg; joints [2.097, -37.612, 126.365, -147.061, 73.323, 69.018, 139.805]
  MoveL 451 to (-197.85, 234.16, -4.14) mm, rotated rx 168.34 ry -27.93 rz 23.78 deg; joints [2.302, -37.607, 126.344, -146.852, 73.312, 69.005, 139.805]
  Set speed (38.1 mm/s)
  MoveL 452 to (-197.89, 234.16, -3.98) mm, rotated rx 168.34 ry -27.93 rz 23.79 deg; joints [2.31, -37.604, 126.343, -146.846, 73.314, 69.004, 139.799]
  MoveL 453 to (-198.05, 233.84, -3.7) mm, rotated rx 168.3 ry -27.91 rz 23.85 deg; joints [2.32, -37.607, 126.352, -146.85, 73.324, 68.983, 139.738]
  Set speed (76.2 mm/s)
  MoveL 454 to (-198.05, 231.3, -3.7) mm, rotated rx 168.14 ry -27.85 rz 24.2 deg; joints [2.307, -37.712, 126.437, -146.93, 73.326, 68.847, 139.429]
  Set speed (38.1 mm/s)
  MoveL 455 to (-197.89, 230.99, -3.98) mm, rotated rx 168.14 ry -27.85 rz 24.21 deg; joints [2.293, -37.735, 126.449, -146.946, 73.317, 68.835, 139.413]
  MoveL 456 to (-197.85, 230.99, -4.14) mm, rotated rx 168.14 ry -27.85 rz 24.21 deg; joints [2.286, -37.738, 126.45, -146.952, 73.315, 68.836, 139.419]
  Set speed (76.2 mm/s)
  MoveL 457 to (-197.85, 230.99, -8.4) mm, rotated rx 168.14 ry -27.85 rz 24.21 deg; joints [2.08, -37.743, 126.471, -147.161, 73.326, 68.849, 139.419]
  MoveL 458 to (-200.15, 230.99, -8.41) mm, rotated rx 167.97 ry -27.78 rz 24.57 deg; joints [2.065, -37.593, 126.473, -147.276, 73.473, 68.803, 139.091]
  MoveL 459 to (-206.05, 230.99, -11.57) mm, rotated rx 167.55 ry -27.61 rz 25.48 deg; joints [1.875, -37.212, 126.489, -147.722, 73.853, 68.699, 138.266]
  MoveL 460 to (-201.08, 230.99, -20.25) mm, rotated rx 167.9 ry -27.75 rz 24.72 deg; joints [1.487, -37.544, 126.525, -147.903, 73.56, 68.817, 138.96]
  MoveL 461 to (-201.08, 227.81, -20.25) mm, rotated rx 167.7 ry -27.67 rz 25.15 deg; joints [1.469, -37.673, 126.633, -148.01, 73.565, 68.649, 138.567]
  MoveL 462 to (-206.05, 227.81, -11.57) mm, rotated rx 167.35 ry -27.52 rz 25.92 deg; joints [1.856, -37.34, 126.598, -147.832, 73.859, 68.532, 137.872]
  MoveL 463 to (-200.15, 227.81, -8.41) mm, rotated rx 167.77 ry -27.7 rz 25 deg; joints [2.047, -37.722, 126.581, -147.382, 73.477, 68.635, 138.698]
  MoveL 464 to (-197.85, 227.81, -8.4) mm, rotated rx 167.94 ry -27.77 rz 24.64 deg; joints [2.062, -37.873, 126.578, -147.265, 73.33, 68.68, 139.027]
  MoveL 465 to (-197.85, 227.81, -4.14) mm, rotated rx 167.94 ry -27.77 rz 24.64 deg; joints [2.268, -37.868, 126.557, -147.056, 73.319, 68.666, 139.027]
  Set speed (38.1 mm/s)
  MoveL 466 to (-197.89, 227.81, -3.98) mm, rotated rx 167.93 ry -27.77 rz 24.65 deg; joints [2.276, -37.865, 126.557, -147.05, 73.321, 68.665, 139.021]
  MoveL 467 to (-198.05, 227.49, -3.7) mm, rotated rx 167.9 ry -27.75 rz 24.72 deg; joints [2.286, -37.867, 126.566, -147.055, 73.331, 68.644, 138.958]
  Set speed (76.2 mm/s)
  MoveL 468 to (-198.05, 224.95, -3.7) mm, rotated rx 167.74 ry -27.69 rz 25.07 deg; joints [2.272, -37.971, 126.653, -147.141, 73.335, 68.508, 138.64]
  Set speed (38.1 mm/s)
  MoveL 469 to (-197.89, 224.64, -3.98) mm, rotated rx 167.73 ry -27.68 rz 25.09 deg; joints [2.258, -37.994, 126.665, -147.157, 73.326, 68.495, 138.622]
  MoveL 470 to (-197.85, 224.64, -4.14) mm, rotated rx 167.73 ry -27.68 rz 25.08 deg; joints [2.25, -37.997, 126.666, -147.163, 73.324, 68.496, 138.629]
  Set speed (76.2 mm/s)
  MoveL 471 to (-197.85, 224.64, -8.4) mm, rotated rx 167.73 ry -27.68 rz 25.08 deg; joints [2.044, -38.001, 126.686, -147.373, 73.335, 68.509, 138.629]
  MoveL 472 to (-200.15, 224.64, -8.41) mm, rotated rx 167.56 ry -27.61 rz 25.45 deg; joints [2.029, -37.851, 126.689, -147.491, 73.483, 68.465, 138.299]
  MoveL 473 to (-206.05, 224.64, -11.57) mm, rotated rx 167.14 ry -27.43 rz 26.36 deg; joints [1.836, -37.468, 126.708, -147.945, 73.866, 68.365, 137.471]
  MoveL 474 to (-201.08, 224.64, -20.25) mm, rotated rx 167.5 ry -27.58 rz 25.59 deg; joints [1.449, -37.801, 126.742, -148.12, 73.57, 68.48, 138.168]
  MoveL 475 to (-201.08, 221.46, -20.25) mm, rotated rx 167.29 ry -27.5 rz 26.04 deg; joints [1.43, -37.928, 126.851, -148.234, 73.577, 68.31, 137.762]
  MoveL 476 to (-206.05, 221.46, -11.57) mm, rotated rx 166.94 ry -27.34 rz 26.8 deg; joints [1.816, -37.594, 126.82, -148.062, 73.874, 68.198, 137.065]
  MoveL 477 to (-200.15, 221.46, -8.41) mm, rotated rx 167.36 ry -27.53 rz 25.89 deg; joints [2.01, -37.978, 126.799, -147.604, 73.49, 68.296, 137.893]
  MoveL 478 to (-197.85, 221.46, -8.4) mm, rotated rx 167.53 ry -27.6 rz 25.53 deg; joints [2.025, -38.129, 126.795, -147.484, 73.341, 68.339, 138.224]
  MoveL 479 to (-197.85, 221.46, -4.14) mm, rotated rx 167.53 ry -27.6 rz 25.53 deg; joints [2.232, -38.125, 126.775, -147.274, 73.33, 68.325, 138.224]
  Set speed (38.1 mm/s)
  MoveL 480 to (-197.89, 221.46, -3.98) mm, rotated rx 167.52 ry -27.6 rz 25.53 deg; joints [2.239, -38.122, 126.774, -147.269, 73.333, 68.324, 138.218]
  MoveL 481 to (-198.05, 221.14, -3.7) mm, rotated rx 167.49 ry -27.58 rz 25.6 deg; joints [2.249, -38.124, 126.784, -147.275, 73.343, 68.303, 138.154]
  Set speed (76.2 mm/s)
  MoveL 482 to (-198.05, 218.6, -3.7) mm, rotated rx 167.32 ry -27.51 rz 25.97 deg; joints [2.234, -38.226, 126.872, -147.367, 73.349, 68.166, 137.825]
  Set speed (38.1 mm/s)
  MoveL 483 to (-197.89, 218.29, -3.98) mm, rotated rx 167.31 ry -27.51 rz 25.99 deg; joints [2.22, -38.249, 126.884, -147.384, 73.34, 68.153, 137.806]
  MoveL 484 to (-197.85, 218.29, -4.14) mm, rotated rx 167.32 ry -27.51 rz 25.98 deg; joints [2.212, -38.252, 126.885, -147.389, 73.338, 68.154, 137.812]
  Set speed (76.2 mm/s)
  MoveL 485 to (-197.85, 218.29, -8.4) mm, rotated rx 167.32 ry -27.51 rz 25.98 deg; joints [2.006, -38.256, 126.906, -147.6, 73.349, 68.168, 137.812]
  MoveL 486 to (-200.15, 218.29, -8.41) mm, rotated rx 167.15 ry -27.43 rz 26.34 deg; joints [1.99, -38.105, 126.91, -147.721, 73.498, 68.125, 137.482]
  MoveL 487 to (-206.05, 218.29, -11.57) mm, rotated rx 166.73 ry -27.25 rz 27.25 deg; joints [1.795, -37.719, 126.932, -148.184, 73.883, 68.03, 136.652]
  MoveL 488 to (-201.08, 218.29, -20.25) mm, rotated rx 167.08 ry -27.4 rz 26.49 deg; joints [1.409, -38.055, 126.962, -148.352, 73.585, 68.14, 137.35]
  MoveL 489 to (-201.08, 215.11, -20.25) mm, rotated rx 166.87 ry -27.31 rz 26.95 deg; joints [1.388, -38.18, 127.074, -148.474, 73.594, 67.97, 136.931]
  MoveL 490 to (-206.05, 215.11, -11.57) mm, rotated rx 166.52 ry -27.15 rz 27.71 deg; joints [1.774, -37.844, 127.045, -148.309, 73.893, 67.862, 136.233]
  MoveL 491 to (-200.15, 215.11, -8.41) mm, rotated rx 166.94 ry -27.34 rz 26.8 deg; joints [1.969, -38.23, 127.022, -147.842, 73.507, 67.955, 137.063]
  MoveL 492 to (-197.85, 215.11, -8.4) mm, rotated rx 167.1 ry -27.41 rz 26.44 deg; joints [1.986, -38.383, 127.017, -147.719, 73.358, 67.996, 137.394]
  MoveL 493 to (-197.85, 215.11, -4.14) mm, rotated rx 167.1 ry -27.41 rz 26.44 deg; joints [2.192, -38.378, 126.996, -147.509, 73.347, 67.983, 137.394]
  Set speed (38.1 mm/s)
  MoveL 494 to (-197.89, 215.11, -3.98) mm, rotated rx 167.1 ry -27.41 rz 26.45 deg; joints [2.2, -38.375, 126.996, -147.503, 73.349, 67.982, 137.388]
  MoveL 495 to (-198.05, 214.79, -3.7) mm, rotated rx 167.07 ry -27.4 rz 26.52 deg; joints [2.21, -38.377, 127.006, -147.51, 73.36, 67.961, 137.323]
  Set speed (76.2 mm/s)
  MoveL 496 to (-198.05, 212.26, -3.7) mm, rotated rx 166.9 ry -27.32 rz 26.89 deg; joints [2.193, -38.477, 127.096, -147.609, 73.368, 67.823, 136.983]
  Set speed (38.1 mm/s)
  MoveL 497 to (-197.89, 211.94, -3.98) mm, rotated rx 166.89 ry -27.32 rz 26.91 deg; joints [2.179, -38.5, 127.108, -147.627, 73.359, 67.81, 136.963]
  MoveL 498 to (-197.85, 211.94, -4.14) mm, rotated rx 166.89 ry -27.32 rz 26.91 deg; joints [2.171, -38.503, 127.109, -147.632, 73.357, 67.811, 136.97]
  Set speed (76.2 mm/s)
  MoveL 499 to (-197.85, 211.94, -8.4) mm, rotated rx 166.89 ry -27.32 rz 26.91 deg; joints [1.965, -38.508, 127.129, -147.843, 73.368, 67.824, 136.97]
  MoveL 500 to (-200.15, 211.94, -8.41) mm, rotated rx 166.72 ry -27.24 rz 27.27 deg; joints [1.948, -38.355, 127.135, -147.967, 73.517, 67.784, 136.638]
  MoveL 501 to (-206.05, 211.94, -11.57) mm, rotated rx 166.31 ry -27.05 rz 28.18 deg; joints [1.751, -37.967, 127.159, -148.438, 73.904, 67.693, 135.807]
  MoveL 502 to (-201.08, 211.94, -20.25) mm, rotated rx 166.66 ry -27.21 rz 27.41 deg; joints [1.366, -38.304, 127.186, -148.601, 73.604, 67.799, 136.506]
  MoveL 503 to (-201.08, 208.76, -20.25) mm, rotated rx 166.44 ry -27.11 rz 27.89 deg; joints [1.343, -38.428, 127.3, -148.731, 73.616, 67.628, 136.074]
  MoveL 504 to (-206.05, 208.76, -11.57) mm, rotated rx 166.1 ry -26.95 rz 28.65 deg; joints [1.728, -38.09, 127.275, -148.572, 73.917, 67.524, 135.375]
  MoveL 505 to (-200.15, 208.76, -8.41) mm, rotated rx 166.51 ry -27.14 rz 27.74 deg; joints [1.926, -38.479, 127.249, -148.097, 73.529, 67.612, 136.206]
  MoveL 506 to (-197.85, 208.76, -8.4) mm, rotated rx 166.67 ry -27.22 rz 27.38 deg; joints [1.943, -38.632, 127.243, -147.97, 73.379, 67.652, 136.538]
  MoveL 507 to (-197.85, 208.76, -4.14) mm, rotated rx 166.67 ry -27.22 rz 27.38 deg; joints [2.15, -38.627, 127.223, -147.76, 73.368, 67.639, 136.538]
  Set speed (38.1 mm/s)
  MoveL 508 to (-197.89, 208.76, -3.98) mm, rotated rx 166.67 ry -27.22 rz 27.39 deg; joints [2.157, -38.624, 127.222, -147.754, 73.371, 67.637, 136.532]
  MoveL 509 to (-198.05, 208.45, -3.7) mm, rotated rx 166.64 ry -27.2 rz 27.46 deg; joints [2.167, -38.626, 127.232, -147.763, 73.382, 67.617, 136.465]
  Set speed (76.2 mm/s)
  MoveL 510 to (-198.05, 205.91, -3.7) mm, rotated rx 166.46 ry -27.12 rz 27.84 deg; joints [2.149, -38.724, 127.324, -147.868, 73.392, 67.479, 136.115]
  Set speed (38.1 mm/s)
  MoveL 511 to (-197.89, 205.59, -3.98) mm, rotated rx 166.45 ry -27.12 rz 27.86 deg; joints [2.135, -38.748, 127.337, -147.887, 73.383, 67.465, 136.093]
  MoveL 512 to (-197.85, 205.59, -4.14) mm, rotated rx 166.45 ry -27.12 rz 27.86 deg; joints [2.127, -38.751, 127.337, -147.892, 73.381, 67.466, 136.1]
  Set speed (76.2 mm/s)
  MoveL 513 to (-197.85, 205.59, -8.4) mm, rotated rx 166.45 ry -27.12 rz 27.86 deg; joints [1.92, -38.755, 127.357, -148.103, 73.391, 67.479, 136.1]
  MoveL 514 to (-200.15, 205.59, -8.41) mm, rotated rx 166.29 ry -27.04 rz 28.22 deg; joints [1.903, -38.601, 127.364, -148.231, 73.542, 67.441, 135.768]
  MoveL 515 to (-206.05, 205.59, -11.57) mm, rotated rx 165.88 ry -26.84 rz 29.13 deg; joints [1.705, -38.211, 127.391, -148.71, 73.931, 67.355, 134.936]
  MoveL 516 to (-201.08, 205.59, -20.25) mm, rotated rx 166.22 ry -27.01 rz 28.36 deg; joints [1.32, -38.55, 127.416, -148.866, 73.629, 67.457, 135.636]
  MoveL 517 to (-201.08, 202.41, -20.25) mm, rotated rx 166 ry -26.9 rz 28.85 deg; joints [1.295, -38.672, 127.532, -149.006, 73.643, 67.285, 135.19]
  MoveL 518 to (-206.05, 202.41, -11.57) mm, rotated rx 165.66 ry -26.73 rz 29.61 deg; joints [1.68, -38.332, 127.509, -148.852, 73.946, 67.185, 134.49]
  MoveL 519 to (-200.15, 202.41, -8.41) mm, rotated rx 166.07 ry -26.93 rz 28.71 deg; joints [1.879, -38.723, 127.481, -148.369, 73.556, 67.269, 135.322]
  MoveL 520 to (-197.85, 202.41, -8.4) mm, rotated rx 166.23 ry -27.01 rz 28.34 deg; joints [1.897, -38.877, 127.473, -148.24, 73.405, 67.306, 135.654]
  MoveL 521 to (-197.85, 202.41, -4.14) mm, rotated rx 166.23 ry -27.01 rz 28.34 deg; joints [2.104, -38.873, 127.453, -148.029, 73.395, 67.293, 135.654]
  Set speed (38.1 mm/s)
  MoveL 522 to (-197.89, 202.41, -3.98) mm, rotated rx 166.23 ry -27.01 rz 28.35 deg; joints [2.112, -38.87, 127.453, -148.023, 73.397, 67.292, 135.648]
  MoveL 523 to (-198.05, 202.1, -3.7) mm, rotated rx 166.2 ry -27 rz 28.43 deg; joints [2.121, -38.871, 127.464, -148.033, 73.408, 67.271, 135.58]
  Set speed (76.2 mm/s)
  MoveL 524 to (-198.05, 199.56, -3.7) mm, rotated rx 166.02 ry -26.91 rz 28.82 deg; joints [2.102, -38.968, 127.558, -148.146, 73.42, 67.133, 135.217]
  Set speed (38.1 mm/s)
  MoveL 525 to (-197.89, 199.24, -3.98) mm, rotated rx 166.01 ry -26.9 rz 28.84 deg; joints [2.088, -38.991, 127.57, -148.165, 73.412, 67.119, 135.195]
  MoveL 526 to (-197.85, 199.24, -4.14) mm, rotated rx 166.01 ry -26.9 rz 28.84 deg; joints [2.08, -38.994, 127.571, -148.17, 73.41, 67.12, 135.201]
  Set speed (76.2 mm/s)
  MoveL 527 to (-197.85, 199.24, -8.4) mm, rotated rx 166.01 ry -26.9 rz 28.84 deg; joints [1.873, -38.998, 127.591, -148.381, 73.42, 67.133, 135.201]
  MoveL 528 to (-200.15, 199.24, -8.41) mm, rotated rx 165.85 ry -26.82 rz 29.2 deg; joints [1.855, -38.844, 127.598, -148.512, 73.572, 67.096, 134.869]
  MoveL 529 to (-206.05, 199.24, -11.57) mm, rotated rx 165.44 ry -26.62 rz 30.1 deg; joints [1.654, -38.452, 127.628, -148.999, 73.962, 67.016, 134.037]
  MoveL 530 to (-201.08, 199.24, -20.25) mm, rotated rx 165.78 ry -26.79 rz 29.34 deg; joints [1.27, -38.793, 127.65, -149.15, 73.658, 67.113, 134.737]
  MoveL 531 to (-201.08, 196.06, -20.25) mm, rotated rx 165.56 ry -26.68 rz 29.84 deg; joints [1.244, -38.912, 127.769, -149.299, 73.675, 66.941, 134.277]
  MoveL 532 to (-206.05, 196.06, -11.57) mm, rotated rx 165.22 ry -26.5 rz 30.6 deg; joints [1.628, -38.571, 127.748, -149.151, 73.979, 66.846, 133.578]
  MoveL 533 to (-200.15, 196.06, -8.41) mm, rotated rx 165.62 ry -26.71 rz 29.7 deg; joints [1.829, -38.964, 127.718, -148.66, 73.588, 66.924, 134.409]
  MoveL 534 to (-197.85, 196.06, -8.4) mm, rotated rx 165.78 ry -26.79 rz 29.34 deg; joints [1.848, -39.119, 127.709, -148.527, 73.437, 66.959, 134.741]
  MoveL 535 to (-197.85, 196.06, -4.14) mm, rotated rx 165.78 ry -26.79 rz 29.34 deg; joints [2.055, -39.114, 127.69, -148.316, 73.426, 66.946, 134.741]
  Set speed (38.1 mm/s)
  MoveL 536 to (-197.89, 196.06, -3.98) mm, rotated rx 165.78 ry -26.79 rz 29.34 deg; joints [2.063, -39.111, 127.689, -148.311, 73.429, 66.945, 134.735]
  MoveL 537 to (-198.05, 195.75, -3.7) mm, rotated rx 165.75 ry -26.77 rz 29.42 deg; joints [2.072, -39.112, 127.7, -148.321, 73.44, 66.924, 134.665]
  Set speed (76.2 mm/s)
  MoveL 538 to (-198.05, 193.21, -3.7) mm, rotated rx 165.56 ry -26.68 rz 29.83 deg; joints [2.052, -39.208, 127.796, -148.442, 73.454, 66.786, 134.291]
  Set speed (38.1 mm/s)
  MoveL 539 to (-197.89, 192.89, -3.98) mm, rotated rx 165.55 ry -26.68 rz 29.85 deg; joints [2.037, -39.231, 127.809, -148.462, 73.446, 66.771, 134.267]
  MoveL 540 to (-197.85, 192.89, -4.14) mm, rotated rx 165.56 ry -26.68 rz 29.84 deg; joints [2.03, -39.234, 127.81, -148.467, 73.444, 66.772, 134.273]
  Set speed (76.2 mm/s)
  MoveL 541 to (-197.85, 192.89, -8.4) mm, rotated rx 165.56 ry -26.68 rz 29.84 deg; joints [1.822, -39.238, 127.829, -148.679, 73.454, 66.785, 134.273]
  MoveL 542 to (-199.6, 192.89, -8.41) mm, rotated rx 165.43 ry -26.61 rz 30.12 deg; joints [1.807, -39.12, 127.836, -148.781, 73.569, 66.759, 134.021]
  MoveL 543 to (-206.05, 192.89, -11.57) mm, rotated rx 164.99 ry -26.38 rz 31.1 deg; joints [1.6, -38.689, 127.87, -149.307, 73.997, 66.676, 133.111]
  MoveL 544 to (-201.08, 192.89, -20.25) mm, rotated rx 165.33 ry -26.56 rz 30.35 deg; joints [1.217, -39.031, 127.889, -149.453, 73.692, 66.768, 133.809]
  MoveL 545 to (-201.08, 189.71, -20.25) mm, rotated rx 165.1 ry -26.44 rz 30.86 deg; joints [1.189, -39.149, 128.011, -149.612, 73.711, 66.595, 133.334]
  MoveL 546 to (-206.05, 189.71, -11.57) mm, rotated rx 164.77 ry -26.26 rz 31.61 deg; joints [1.572, -38.806, 127.993, -149.469, 74.017, 66.505, 132.637]
  MoveL 547 to (-199.6, 189.71, -8.41) mm, rotated rx 165.2 ry -26.49 rz 30.63 deg; joints [1.78, -39.238, 127.958, -148.938, 73.588, 66.586, 133.546]
  MoveL 548 to (-197.85, 189.71, -8.4) mm, rotated rx 165.32 ry -26.56 rz 30.36 deg; joints [1.795, -39.357, 127.951, -148.835, 73.473, 66.611, 133.798]
  MoveL 549 to (-197.85, 189.71, -4.14) mm, rotated rx 165.32 ry -26.56 rz 30.36 deg; joints [2.003, -39.352, 127.931, -148.623, 73.463, 66.599, 133.798]
  MoveL 550 to (-197.85, 189.59, -3.66) mm, rotated rx 165.32 ry -26.55 rz 30.38 deg; joints [2.025, -39.357, 127.934, -148.606, 73.462, 66.59, 133.779]
  MoveL 551 to (-197.85, 189.24, -3.31) mm, rotated rx 165.29 ry -26.54 rz 30.44 deg; joints [2.039, -39.369, 127.946, -148.606, 73.464, 66.57, 133.726]
  MoveL 552 to (-197.85, 188.76, -3.19) mm, rotated rx 165.26 ry -26.52 rz 30.52 deg; joints [2.041, -39.387, 127.964, -148.624, 73.466, 66.543, 133.654]
  MoveL 553 to (-197.85, 187.49, -3.19) mm, rotated rx 165.16 ry -26.47 rz 30.72 deg; joints [2.03, -39.434, 128.013, -148.688, 73.474, 66.474, 133.461]
  MoveL 554 to (-197.85, 187.02, -3.31) mm, rotated rx 165.13 ry -26.45 rz 30.8 deg; joints [2.02, -39.451, 128.032, -148.719, 73.478, 66.448, 133.388]
  MoveL 555 to (-197.85, 186.67, -3.66) mm, rotated rx 165.1 ry -26.44 rz 30.86 deg; joints [2, -39.465, 128.047, -148.754, 73.481, 66.43, 133.335]
  MoveL 556 to (-197.85, 186.54, -4.14) mm, rotated rx 165.09 ry -26.43 rz 30.88 deg; joints [1.975, -39.47, 128.054, -148.785, 73.483, 66.424, 133.315]
  MoveL 557 to (-197.85, 186.54, -8.4) mm, rotated rx 165.09 ry -26.43 rz 30.88 deg; joints [1.767, -39.474, 128.074, -148.996, 73.493, 66.437, 133.315]
  MoveL 558 to (-199.6, 186.54, -8.41) mm, rotated rx 164.97 ry -26.37 rz 31.15 deg; joints [1.752, -39.356, 128.081, -149.101, 73.609, 66.413, 133.063]
  MoveL 559 to (-206.05, 186.54, -11.57) mm, rotated rx 164.54 ry -26.13 rz 32.13 deg; joints [1.543, -38.922, 128.117, -149.635, 74.037, 66.335, 132.155]
  MoveL 560 to (-201.08, 186.54, -20.25) mm, rotated rx 164.87 ry -26.31 rz 31.38 deg; joints [1.16, -39.266, 128.134, -149.776, 73.731, 66.422, 132.852]
  MoveL 561 to (-201.08, 183.37, -20.25) mm, rotated rx 164.64 ry -26.19 rz 31.91 deg; joints [1.13, -39.382, 128.258, -149.945, 73.752, 66.249, 132.362]
  MoveL 562 to (-206.05, 183.37, -11.57) mm, rotated rx 164.31 ry -26 rz 32.65 deg; joints [1.512, -39.037, 128.243, -149.807, 74.059, 66.165, 131.666]
  MoveL 563 to (-199.6, 183.37, -8.41) mm, rotated rx 164.74 ry -26.24 rz 31.68 deg; joints [1.723, -39.472, 128.206, -149.269, 73.63, 66.239, 132.573]
  MoveL 564 to (-197.85, 183.37, -8.4) mm, rotated rx 164.86 ry -26.31 rz 31.41 deg; joints [1.738, -39.591, 128.198, -149.163, 73.514, 66.263, 132.825]
  MoveL 565 to (-197.85, 183.37, -4.14) mm, rotated rx 164.86 ry -26.31 rz 31.41 deg; joints [1.946, -39.586, 128.179, -148.951, 73.504, 66.25, 132.825]
  MoveL 566 to (-197.85, 183.24, -3.66) mm, rotated rx 164.85 ry -26.3 rz 31.43 deg; joints [1.969, -39.591, 128.182, -148.934, 73.504, 66.242, 132.805]
  MoveL 567 to (-197.85, 182.89, -3.31) mm, rotated rx 164.82 ry -26.29 rz 31.49 deg; joints [1.982, -39.603, 128.194, -148.936, 73.505, 66.222, 132.75]
  MoveL 568 to (-197.85, 182.41, -3.19) mm, rotated rx 164.79 ry -26.27 rz 31.57 deg; joints [1.984, -39.62, 128.212, -148.955, 73.508, 66.195, 132.676]
  MoveL 569 to (-197.85, 181.14, -3.19) mm, rotated rx 164.69 ry -26.22 rz 31.78 deg; joints [1.972, -39.667, 128.263, -149.024, 73.517, 66.125, 132.477]
  MoveL 570 to (-197.85, 180.67, -3.31) mm, rotated rx 164.66 ry -26.2 rz 31.87 deg; joints [1.962, -39.684, 128.282, -149.056, 73.521, 66.1, 132.401]
  MoveL 571 to (-197.85, 180.32, -3.66) mm, rotated rx 164.63 ry -26.18 rz 31.92 deg; joints [1.941, -39.697, 128.298, -149.093, 73.524, 66.082, 132.346]
  MoveL 572 to (-197.85, 180.19, -4.14) mm, rotated rx 164.62 ry -26.18 rz 31.95 deg; joints [1.917, -39.702, 128.305, -149.123, 73.527, 66.076, 132.326]
  MoveL 573 to (-197.85, 180.19, -8.4) mm, rotated rx 164.62 ry -26.18 rz 31.95 deg; joints [1.708, -39.706, 128.324, -149.335, 73.536, 66.088, 132.326]
  MoveL 574 to (-199.6, 180.19, -8.41) mm, rotated rx 164.5 ry -26.11 rz 32.22 deg; joints [1.692, -39.587, 128.332, -149.442, 73.652, 66.066, 132.075]
  MoveL 575 to (-206.05, 180.19, -11.57) mm, rotated rx 164.08 ry -25.86 rz 33.19 deg; joints [1.481, -39.151, 128.371, -149.984, 74.082, 65.994, 131.17]
  MoveL 576 to (-201.08, 180.19, -20.25) mm, rotated rx 164.4 ry -26.05 rz 32.44 deg; joints [1.099, -39.497, 128.384, -150.12, 73.775, 66.076, 131.864]
  MoveL 577 to (-201.08, 177.02, -20.25) mm, rotated rx 164.16 ry -25.92 rz 32.98 deg; joints [1.067, -39.611, 128.512, -150.3, 73.798, 65.903, 131.359]
  MoveL 578 to (-206.05, 177.02, -11.57) mm, rotated rx 163.84 ry -25.72 rz 33.72 deg; joints [1.449, -39.265, 128.5, -150.167, 74.106, 65.824, 130.666]
  MoveL 579 to (-199.6, 177.02, -8.41) mm, rotated rx 164.26 ry -25.97 rz 32.76 deg; joints [1.661, -39.702, 128.46, -149.621, 73.676, 65.892, 131.569]
  MoveL 580 to (-197.85, 177.02, -8.4) mm, rotated rx 164.38 ry -26.04 rz 32.49 deg; joints [1.677, -39.821, 128.452, -149.513, 73.56, 65.914, 131.82]
  MoveL 581 to (-197.85, 177.02, -4.14) mm, rotated rx 164.38 ry -26.04 rz 32.49 deg; joints [1.886, -39.817, 128.433, -149.301, 73.55, 65.902, 131.82]
  MoveL 582 to (-197.85, 176.89, -3.66) mm, rotated rx 164.37 ry -26.03 rz 32.51 deg; joints [1.908, -39.821, 128.436, -149.285, 73.55, 65.893, 131.799]
  MoveL 583 to (-197.85, 176.54, -3.31) mm, rotated rx 164.34 ry -26.02 rz 32.57 deg; joints [1.922, -39.833, 128.449, -149.287, 73.552, 65.873, 131.743]
  MoveL 584 to (-197.85, 176.06, -3.19) mm, rotated rx 164.31 ry -26 rz 32.65 deg; joints [1.923, -39.85, 128.467, -149.308, 73.555, 65.847, 131.666]
  MoveL 585 to (-197.85, 174.79, -3.19) mm, rotated rx 164.21 ry -25.94 rz 32.87 deg; joints [1.91, -39.896, 128.519, -149.381, 73.565, 65.777, 131.46]
  MoveL 586 to (-197.85, 174.32, -3.31) mm, rotated rx 164.18 ry -25.92 rz 32.96 deg; joints [1.899, -39.913, 128.539, -149.416, 73.569, 65.751, 131.383]
  MoveL 587 to (-197.85, 173.97, -3.66) mm, rotated rx 164.15 ry -25.91 rz 33.02 deg; joints [1.879, -39.926, 128.555, -149.453, 73.573, 65.733, 131.326]
  MoveL 588 to (-197.85, 173.84, -4.14) mm, rotated rx 164.14 ry -25.9 rz 33.04 deg; joints [1.854, -39.931, 128.562, -149.485, 73.575, 65.727, 131.305]
  MoveL 589 to (-197.85, 173.84, -8.4) mm, rotated rx 164.14 ry -25.9 rz 33.04 deg; joints [1.645, -39.935, 128.581, -149.697, 73.585, 65.739, 131.305]
  MoveL 590 to (-199.6, 173.84, -8.41) mm, rotated rx 164.02 ry -25.83 rz 33.31 deg; joints [1.629, -39.815, 128.59, -149.805, 73.701, 65.719, 131.054]
  MoveL 591 to (-206.05, 173.84, -11.57) mm, rotated rx 163.61 ry -25.58 rz 34.27 deg; joints [1.415, -39.377, 128.63, -150.355, 74.131, 65.653, 130.154]
  MoveL 592 to (-201.08, 173.84, -20.25) mm, rotated rx 163.93 ry -25.77 rz 33.53 deg; joints [1.033, -39.724, 128.641, -150.486, 73.823, 65.729, 130.845]
  MoveL 593 to (-201.08, 170.67, -20.25) mm, rotated rx 163.68 ry -25.63 rz 34.09 deg; joints [0.999, -39.836, 128.772, -150.678, 73.849, 65.556, 130.323]
  MoveL 594 to (-206.05, 170.67, -11.57) mm, rotated rx 163.37 ry -25.43 rz 34.82 deg; joints [1.38, -39.489, 128.762, -150.549, 74.157, 65.483, 129.634]
  MoveL 595 to (-199.6, 170.67, -8.41) mm, rotated rx 163.78 ry -25.69 rz 33.87 deg; joints [1.595, -39.928, 128.721, -149.996, 73.727, 65.545, 130.532]
  MoveL 596 to (-197.85, 170.67, -8.4) mm, rotated rx 163.9 ry -25.76 rz 33.6 deg; joints [1.612, -40.048, 128.712, -149.887, 73.611, 65.565, 130.782]
  MoveL 597 to (-197.85, 170.67, -4.14) mm, rotated rx 163.9 ry -25.76 rz 33.6 deg; joints [1.821, -40.044, 128.694, -149.674, 73.601, 65.553, 130.782]
  Set speed (38.1 mm/s)
  MoveL 598 to (-197.89, 170.67, -3.98) mm, rotated rx 163.89 ry -25.76 rz 33.61 deg; joints [1.828, -40.041, 128.693, -149.669, 73.603, 65.552, 130.776]
  MoveL 599 to (-198.05, 170.35, -3.7) mm, rotated rx 163.86 ry -25.73 rz 33.69 deg; joints [1.837, -40.041, 128.706, -149.684, 73.616, 65.532, 130.7]
  Set speed (76.2 mm/s)
  MoveL 600 to (-198.05, 167.81, -3.7) mm, rotated rx 163.66 ry -25.62 rz 34.14 deg; joints [1.81, -40.131, 128.812, -149.84, 73.638, 65.393, 130.275]
  Set speed (38.1 mm/s)
  MoveL 601 to (-197.89, 167.49, -3.98) mm, rotated rx 163.65 ry -25.61 rz 34.17 deg; joints [1.794, -40.153, 128.826, -149.864, 73.631, 65.378, 130.244]
  MoveL 602 to (-197.85, 167.49, -4.14) mm, rotated rx 163.65 ry -25.61 rz 34.17 deg; joints [1.787, -40.156, 128.827, -149.869, 73.628, 65.379, 130.251]
  Set speed (76.2 mm/s)
  MoveL 603 to (-197.85, 167.49, -8.4) mm, rotated rx 163.65 ry -25.61 rz 34.17 deg; joints [1.577, -40.16, 128.845, -150.082, 73.638, 65.391, 130.251]
  MoveL 604 to (-199.6, 167.49, -8.41) mm, rotated rx 163.54 ry -25.54 rz 34.43 deg; joints [1.56, -40.04, 128.854, -150.192, 73.754, 65.372, 130.002]
  MoveL 605 to (-206.05, 167.49, -11.57) mm, rotated rx 163.13 ry -25.28 rz 35.38 deg; joints [1.344, -39.6, 128.896, -150.749, 74.184, 65.313, 129.107]
  MoveL 606 to (-201.08, 167.49, -20.25) mm, rotated rx 163.44 ry -25.48 rz 34.65 deg; joints [0.963, -39.948, 128.905, -150.876, 73.876, 65.383, 129.793]
  MoveL 607 to (-201.08, 164.32, -20.25) mm, rotated rx 163.2 ry -25.32 rz 35.22 deg; joints [0.926, -40.059, 129.039, -151.079, 73.904, 65.21, 129.255]
  MoveL 608 to (-206.05, 164.32, -11.57) mm, rotated rx 162.89 ry -25.12 rz 35.95 deg; joints [1.307, -39.71, 129.031, -150.955, 74.212, 65.143, 128.571]
  MoveL 609 to (-199.6, 164.32, -8.41) mm, rotated rx 163.29 ry -25.38 rz 35 deg; joints [1.524, -40.151, 128.989, -150.395, 73.782, 65.199, 129.463]
  MoveL 610 to (-197.85, 164.32, -8.4) mm, rotated rx 163.4 ry -25.46 rz 34.74 deg; joints [1.541, -40.271, 128.979, -150.284, 73.666, 65.217, 129.711]
  MoveL 611 to (-197.85, 164.32, -4.14) mm, rotated rx 163.4 ry -25.46 rz 34.74 deg; joints [1.751, -40.267, 128.961, -150.071, 73.656, 65.205, 129.711]
  Set speed (38.1 mm/s)
  MoveL 612 to (-197.89, 164.32, -3.98) mm, rotated rx 163.4 ry -25.45 rz 34.75 deg; joints [1.759, -40.264, 128.961, -150.066, 73.659, 65.204, 129.705]
  MoveL 613 to (-198.05, 164, -3.7) mm, rotated rx 163.37 ry -25.43 rz 34.83 deg; joints [1.767, -40.264, 128.974, -150.082, 73.671, 65.184, 129.628]
  Set speed (76.2 mm/s)
  MoveL 614 to (-198.05, 161.46, -3.7) mm, rotated rx 163.17 ry -25.31 rz 35.29 deg; joints [1.738, -40.352, 129.083, -150.249, 73.695, 65.046, 129.189]
  Set speed (38.1 mm/s)
  MoveL 615 to (-197.89, 161.14, -3.98) mm, rotated rx 163.15 ry -25.3 rz 35.33 deg; joints [1.722, -40.375, 129.097, -150.273, 73.688, 65.031, 129.156]
